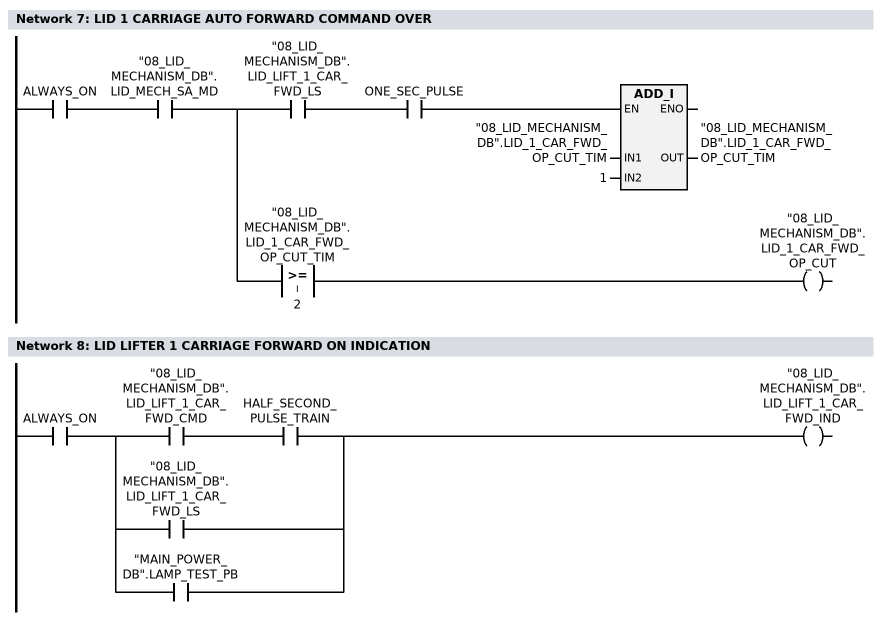
[picture p120: LID_1_MECHANISM networks 7-8]
NETWORK
TITLE = LID 1 CARRIAGE AUTO FORWARD COMMAND OVER
      A     "ALWAYS_ON";
      A     "08_LID_MECHANISM_DB".LID_MECH_SA_MD;
      =     L 0.0;
      A     L 0.0;
      A     "08_LID_MECHANISM_DB".LID_LIFT_1_CAR_FWD_LS;
      A     "ONE_SEC_PULSE";
      JNB   _002;
      L     "08_LID_MECHANISM_DB".LID_1_CAR_FWD_OP_CUT_TIM;
      L     1;
      +I;
      T     "08_LID_MECHANISM_DB".LID_1_CAR_FWD_OP_CUT_TIM;
_002: NOP   0;
      A     L 0.0;
      A(;
      L     "08_LID_MECHANISM_DB".LID_1_CAR_FWD_OP_CUT_TIM;
      L     2;
      >=I;
      );
      =     "08_LID_MECHANISM_DB".LID_1_CAR_FWD_OP_CUT;
NETWORK
TITLE = LID LIFTER 1 CARRIAGE FORWARD ON INDICATION
      A     "ALWAYS_ON";
      A(;
      A     "08_LID_MECHANISM_DB".LID_LIFT_1_CAR_FWD_CMD;
      A     "HALF_SECOND_PULSE_TRAIN";
      O     "08_LID_MECHANISM_DB".LID_LIFT_1_CAR_FWD_LS;
      O     "MAIN_POWER_DB".LAMP_TEST_PB;
      );
      =     "08_LID_MECHANISM_DB".LID_LIFT_1_CAR_FWD_IND;
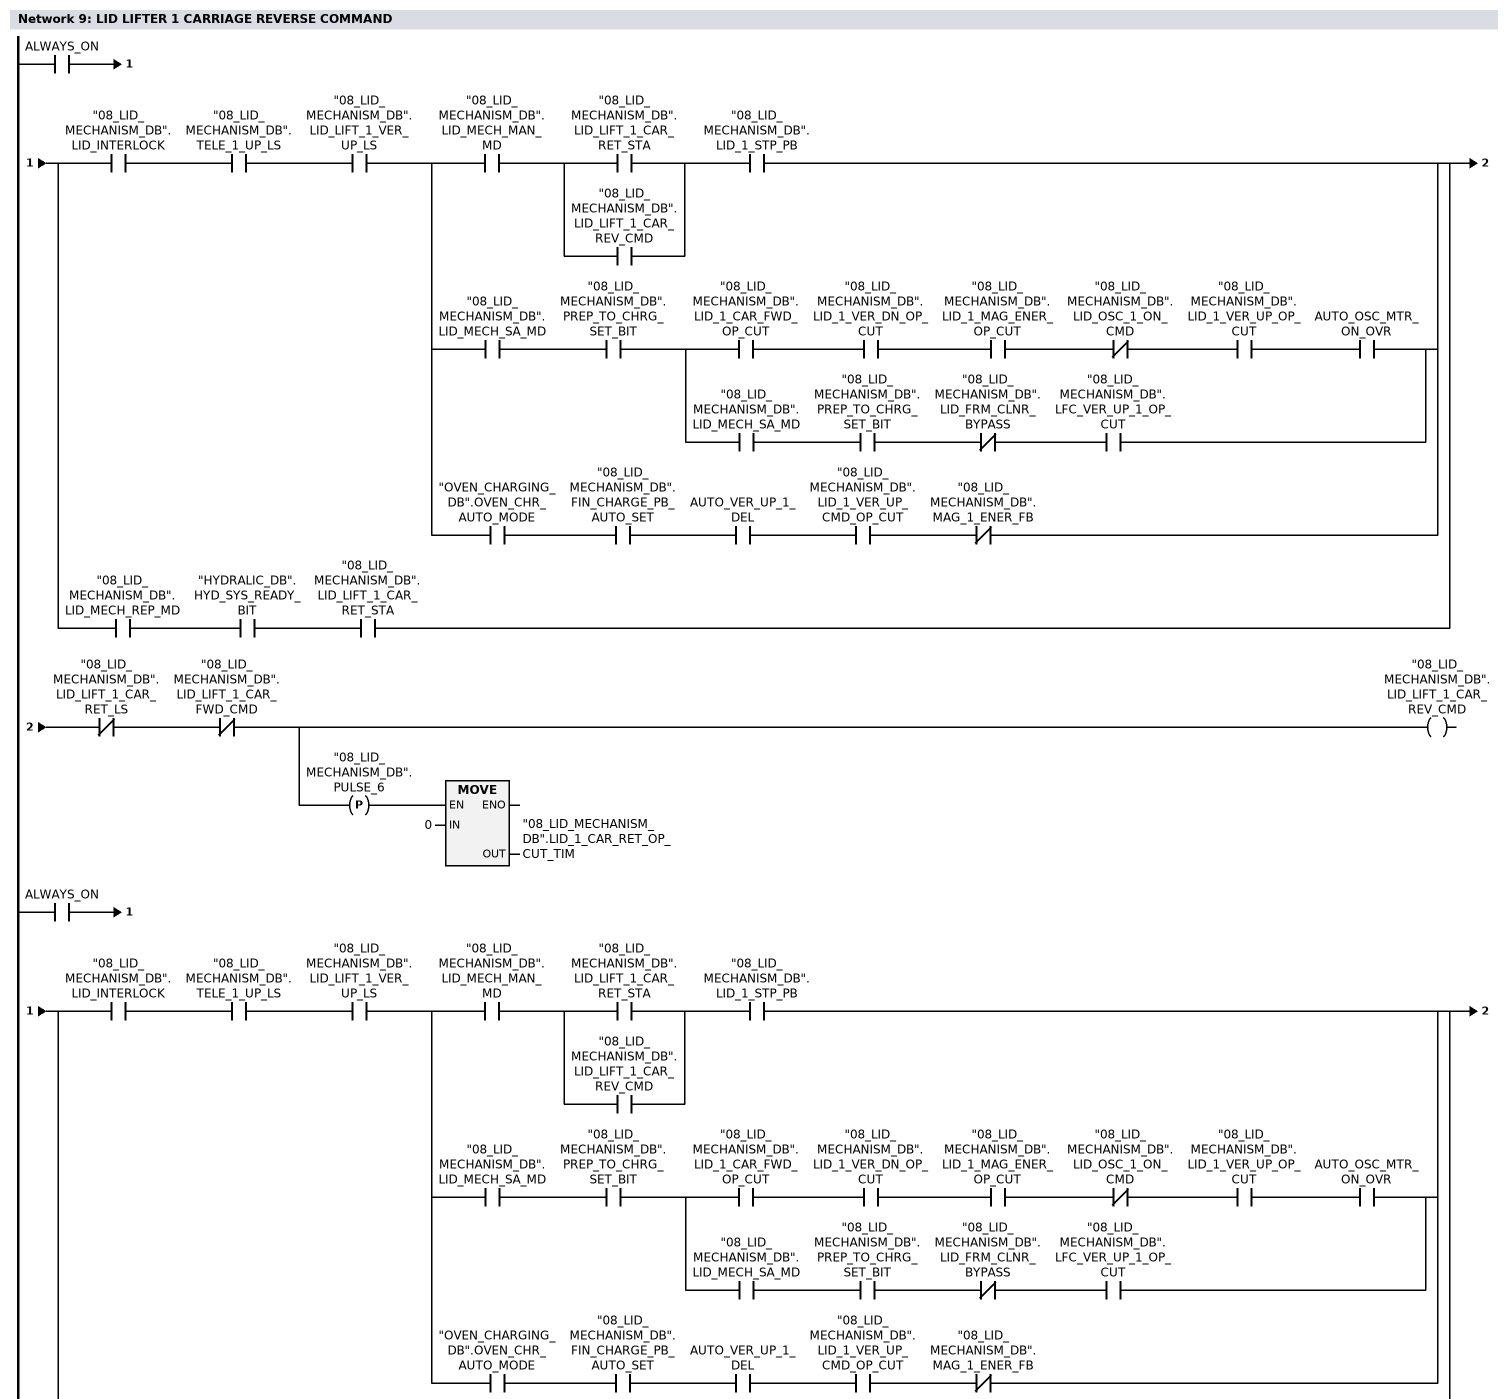
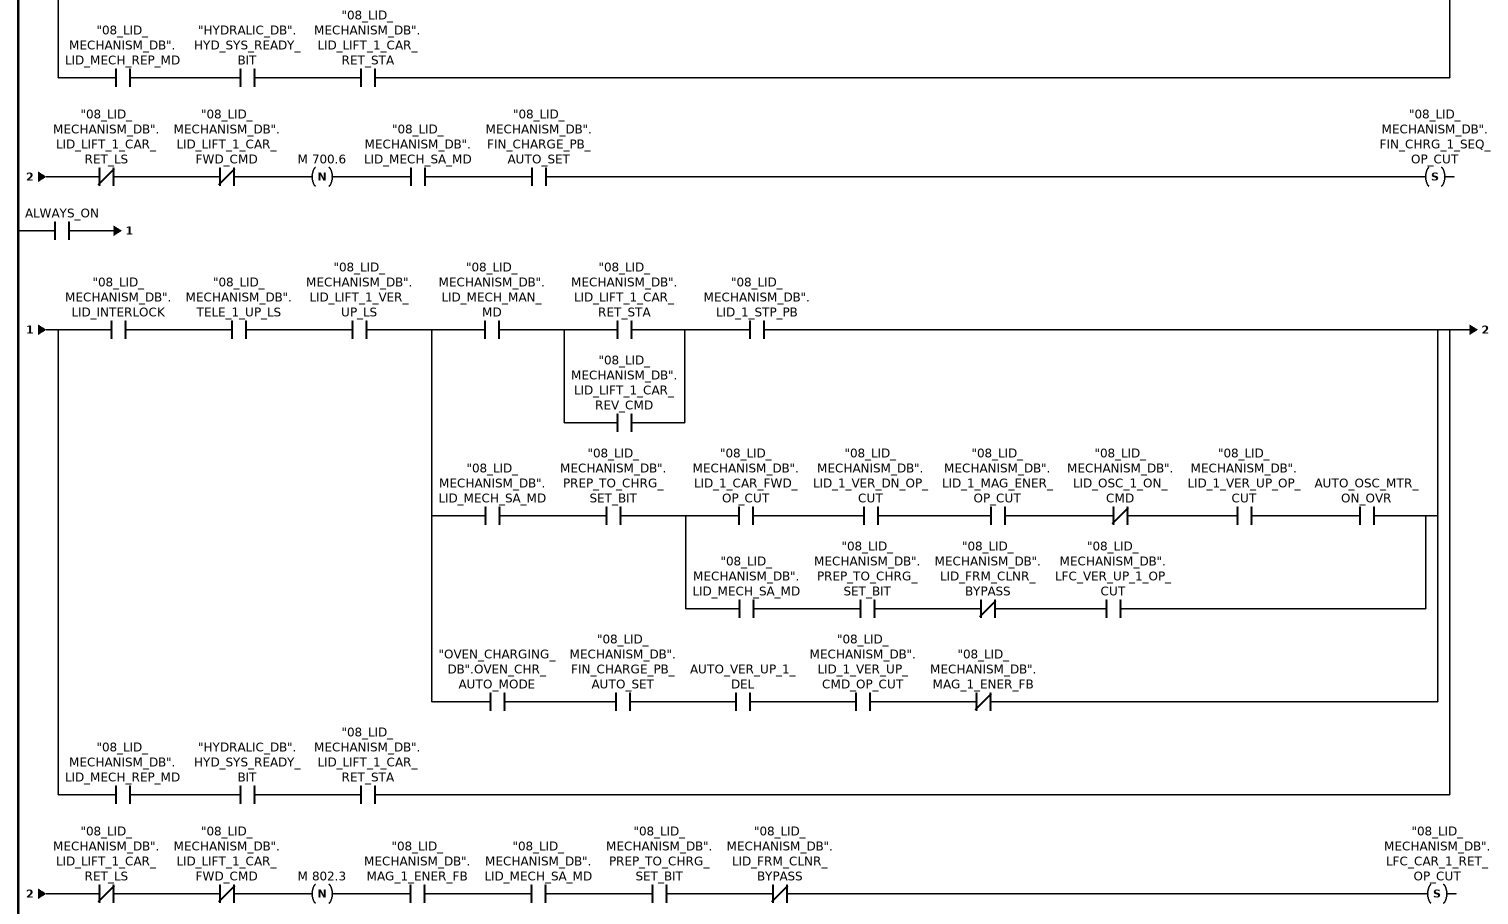
NETWORK
TITLE = LID LIFTER 1 CARRIAGE REVERSE COMMAND
      A     "ALWAYS_ON";
      A(;
      A     "08_LID_MECHANISM_DB".LID_INTERLOCK;
      A     "08_LID_MECHANISM_DB".TELE_1_UP_LS;
      A     "08_LID_MECHANISM_DB".LID_LIFT_1_VER_UP_LS;
      A(;
      A     "08_LID_MECHANISM_DB".LID_MECH_MAN_MD;
      A(;
      O     "08_LID_MECHANISM_DB".LID_LIFT_1_CAR_RET_STA;
      O     "08_LID_MECHANISM_DB".LID_LIFT_1_CAR_REV_CMD;
      );
      A     "08_LID_MECHANISM_DB".LID_1_STP_PB;
      O;
      A     "08_LID_MECHANISM_DB".LID_MECH_SA_MD;
      A     "08_LID_MECHANISM_DB".PREP_TO_CHRG_SET_BIT;
      A(;
      A     "08_LID_MECHANISM_DB".LID_1_CAR_FWD_OP_CUT;
      A     "08_LID_MECHANISM_DB".LID_1_VER_DN_OP_CUT;
      A     "08_LID_MECHANISM_DB".LID_1_MAG_ENER_OP_CUT;
      AN    "08_LID_MECHANISM_DB".LID_OSC_1_ON_CMD;
      A     "08_LID_MECHANISM_DB".LID_1_VER_UP_OP_CUT;
      A     "AUTO_OSC_MTR_ON_OVR";
      O;
      A     "08_LID_MECHANISM_DB".LID_MECH_SA_MD;
      A     "08_LID_MECHANISM_DB".PREP_TO_CHRG_SET_BIT;
      AN    "08_LID_MECHANISM_DB".LID_FRM_CLNR_BYPASS;
      A     "08_LID_MECHANISM_DB".LFC_VER_UP_1_OP_CUT;
      );
      O;
      A     "OVEN_CHARGING_DB".OVEN_CHR_AUTO_MODE;
      A     "08_LID_MECHANISM_DB".FIN_CHARGE_PB_AUTO_SET;
      A     "AUTO_VER_UP_1_DEL";
      A     "08_LID_MECHANISM_DB".LID_1_VER_UP_CMD_OP_CUT;
      AN    "08_LID_MECHANISM_DB".MAG_1_ENER_FB;
      );
      O;
      A     "08_LID_MECHANISM_DB".LID_MECH_REP_MD;
      A     "HYDRALIC_DB".HYD_SYS_READY_BIT;
      A     "08_LID_MECHANISM_DB".LID_LIFT_1_CAR_RET_STA;
      );
      AN    "08_LID_MECHANISM_DB".LID_LIFT_1_CAR_RET_LS;
      AN    "08_LID_MECHANISM_DB".LID_LIFT_1_CAR_FWD_CMD;
      =     L 0.0;
      A     L 0.0;
      BLD   102;
      =     "08_LID_MECHANISM_DB".LID_LIFT_1_CAR_REV_CMD;
      A     L 0.0;
      FP    "08_LID_MECHANISM_DB".PULSE_6;
      JNB   _003;
      L     0;
      T     "08_LID_MECHANISM_DB".LID_1_CAR_RET_OP_CUT_TIM;
_003: NOP   0;
      A(;
      A     L 0.0;
      FN    M 700.6;
      );
      A     "08_LID_MECHANISM_DB".LID_MECH_SA_MD;
      A     "08_LID_MECHANISM_DB".FIN_CHARGE_PB_AUTO_SET;
      S     "08_LID_MECHANISM_DB".FIN_CHRG_1_SEQ_OP_CUT;
      A(;
      A     L 0.0;
      FN    M 802.3;
      );
      A     "08_LID_MECHANISM_DB".MAG_1_ENER_FB;
      A     "08_LID_MECHANISM_DB".LID_MECH_SA_MD;
      A     "08_LID_MECHANISM_DB".PREP_TO_CHRG_SET_BIT;
      AN    "08_LID_MECHANISM_DB".LID_FRM_CLNR_BYPASS;
      S     "08_LID_MECHANISM_DB".LFC_CAR_1_RET_OP_CUT;
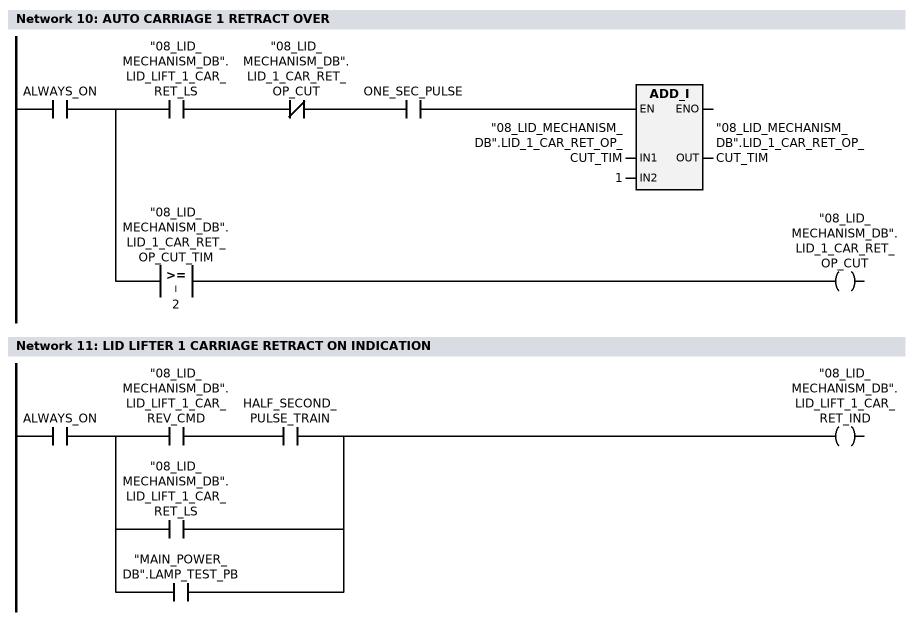
NETWORK
TITLE = AUTO CARRIAGE 1 RETRACT OVER
      A     "ALWAYS_ON";
      =     L 0.0;
      A     L 0.0;
      A     "08_LID_MECHANISM_DB".LID_LIFT_1_CAR_RET_LS;
      AN    "08_LID_MECHANISM_DB".LID_1_CAR_RET_OP_CUT;
      A     "ONE_SEC_PULSE";
      JNB   _004;
      L     "08_LID_MECHANISM_DB".LID_1_CAR_RET_OP_CUT_TIM;
      L     1;
      +I;
      T     "08_LID_MECHANISM_DB".LID_1_CAR_RET_OP_CUT_TIM;
_004: NOP   0;
      A     L 0.0;
      A(;
      L     "08_LID_MECHANISM_DB".LID_1_CAR_RET_OP_CUT_TIM;
      L     2;
      >=I;
      );
      =     "08_LID_MECHANISM_DB".LID_1_CAR_RET_OP_CUT;
NETWORK
TITLE = LID LIFTER 1 CARRIAGE RETRACT ON INDICATION
      A     "ALWAYS_ON";
      A(;
      A     "08_LID_MECHANISM_DB".LID_LIFT_1_CAR_REV_CMD;
      A     "HALF_SECOND_PULSE_TRAIN";
      O     "08_LID_MECHANISM_DB".LID_LIFT_1_CAR_RET_LS;
      O     "MAIN_POWER_DB".LAMP_TEST_PB;
      );
      =     "08_LID_MECHANISM_DB".LID_LIFT_1_CAR_RET_IND;
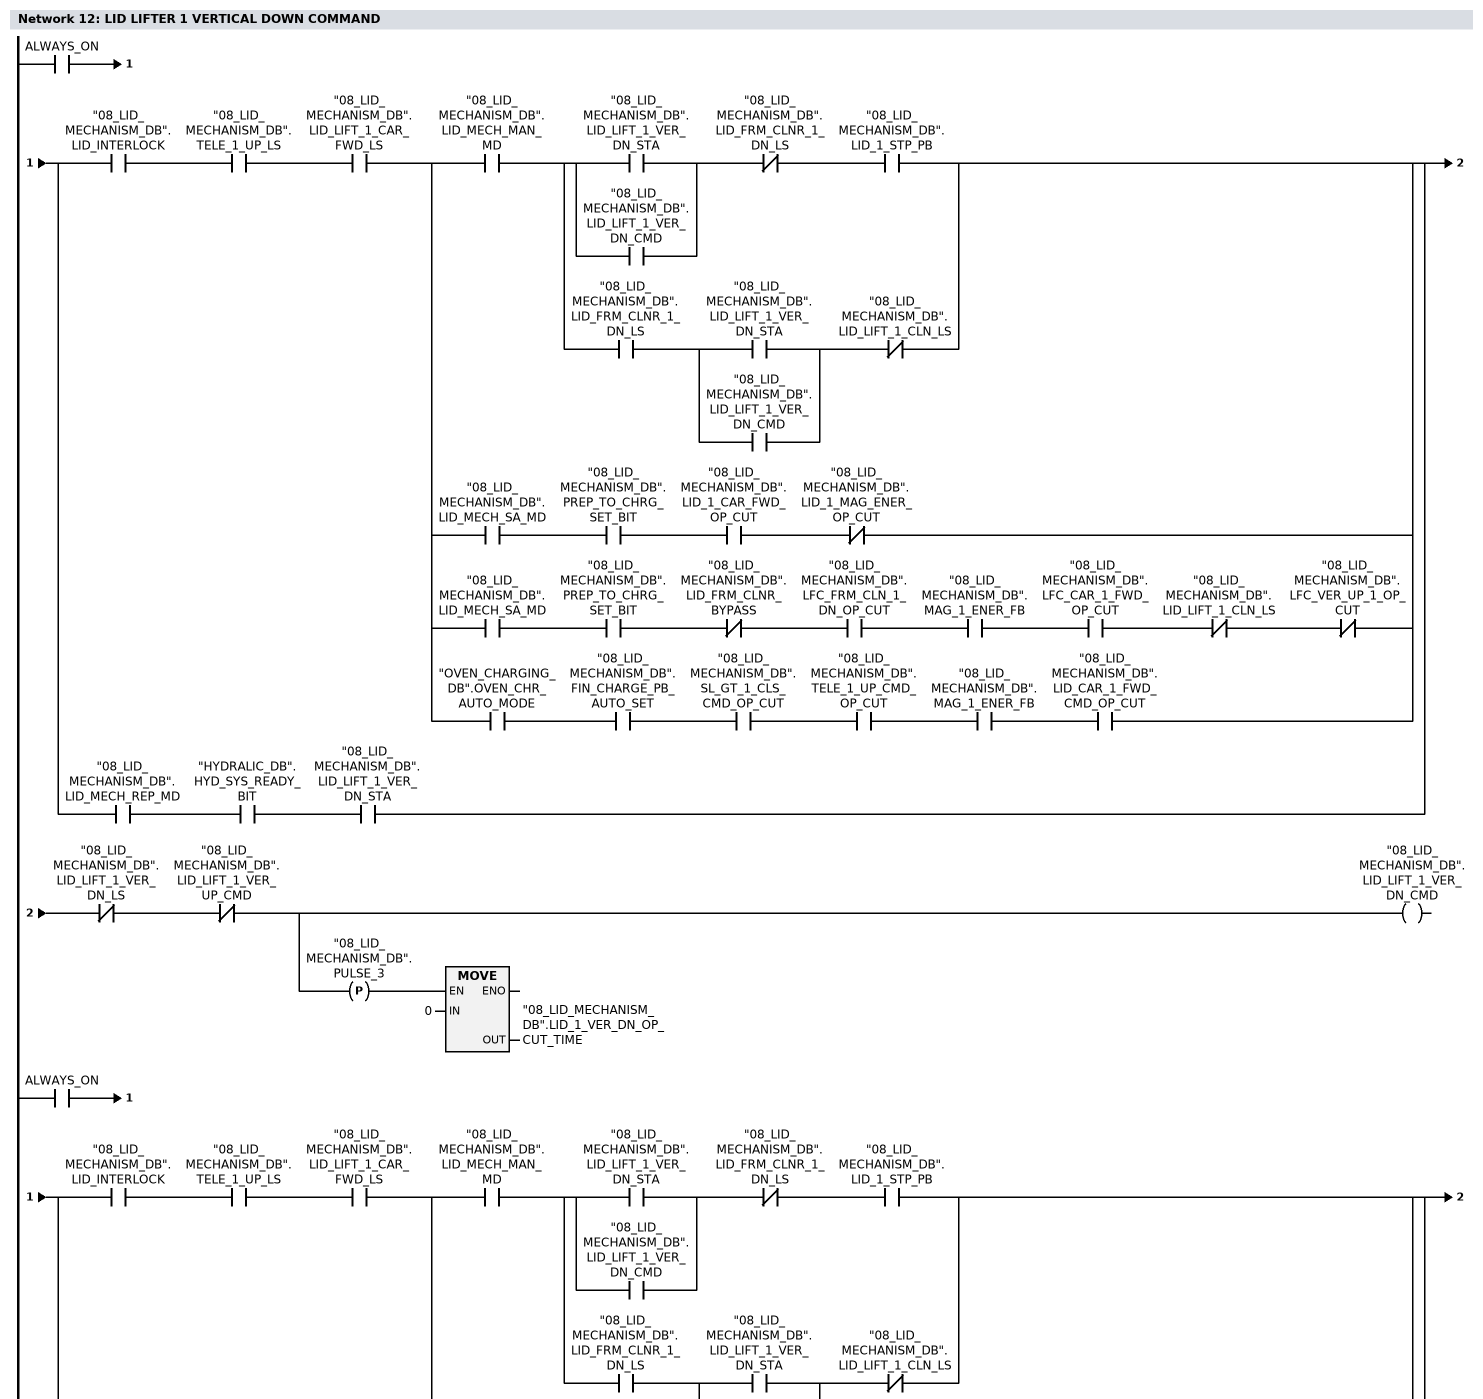
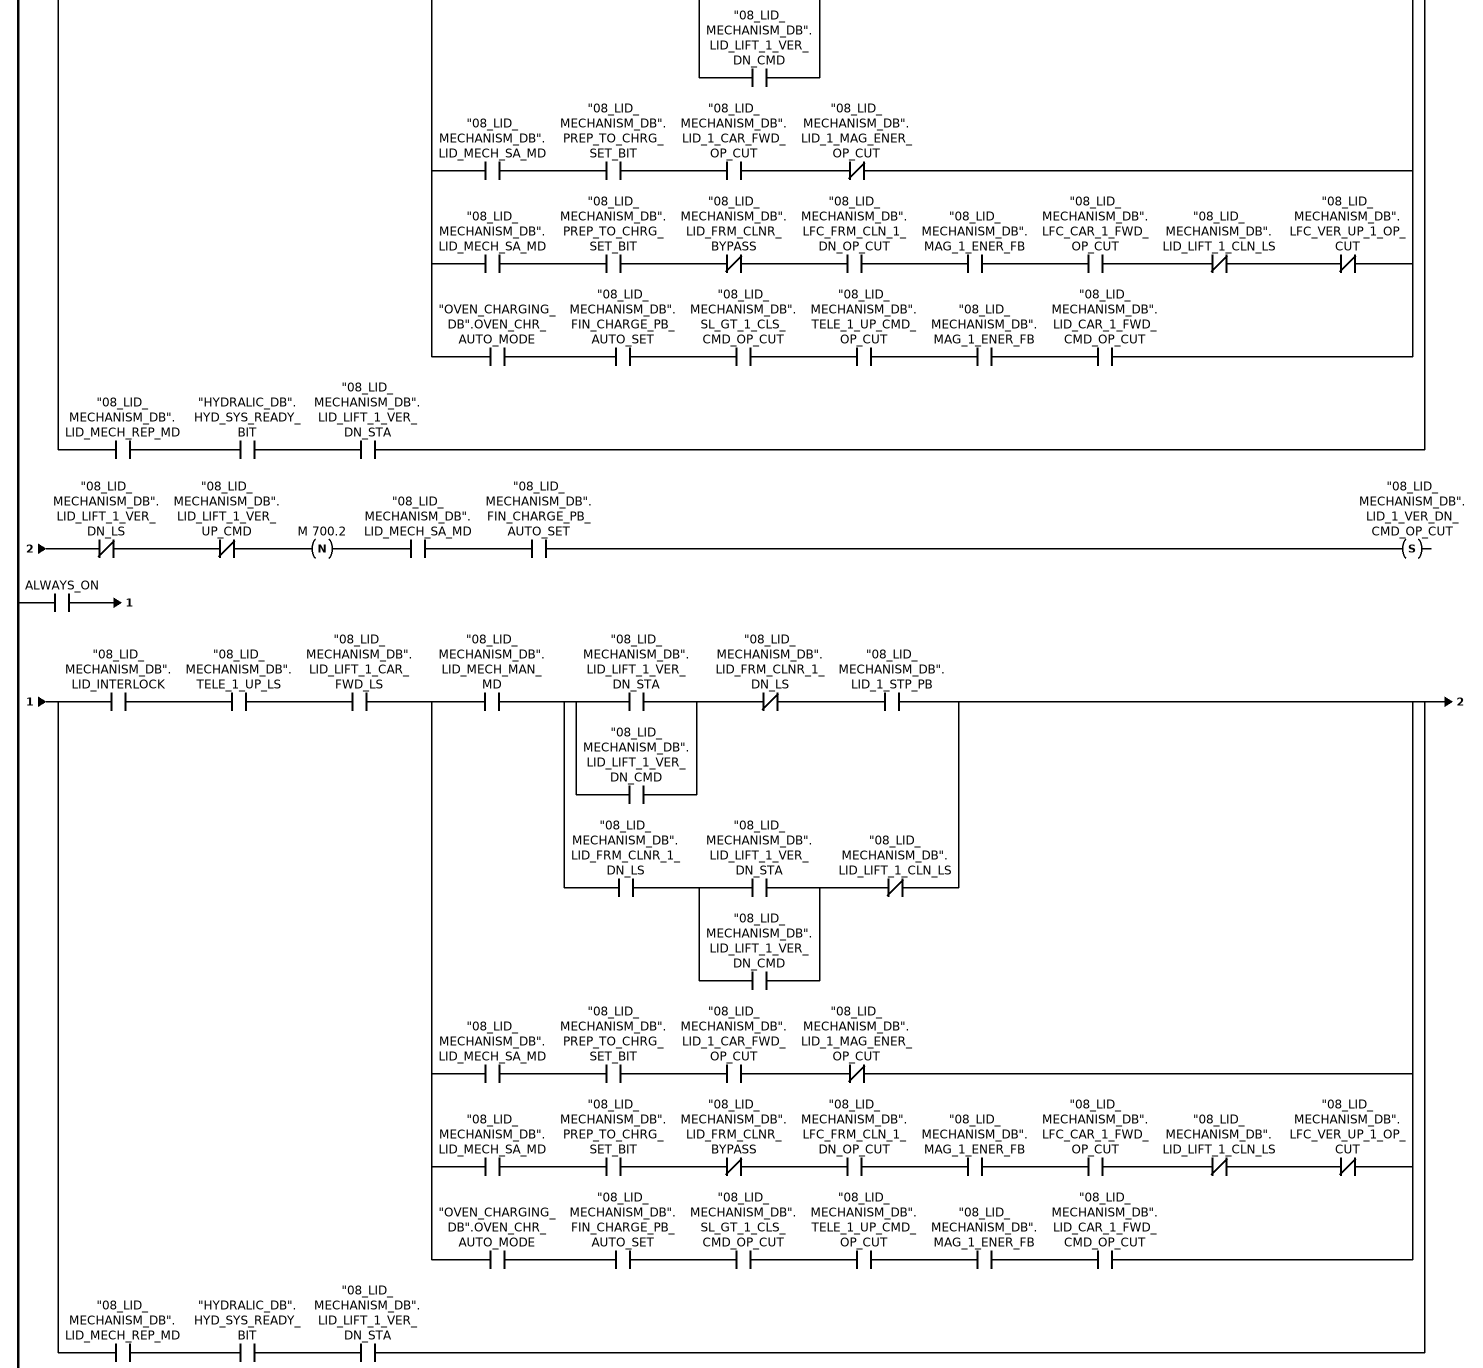
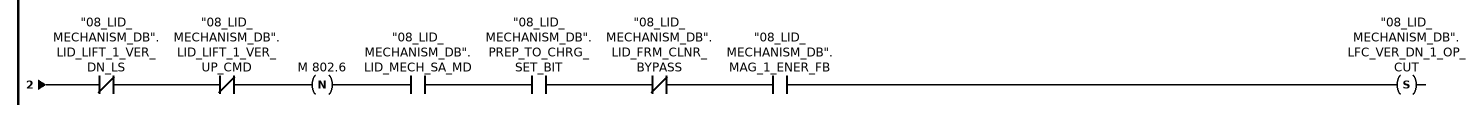
NETWORK
TITLE = LID LIFTER 1 VERTICAL DOWN COMMAND
      A     "ALWAYS_ON";
      A(;
      A     "08_LID_MECHANISM_DB".LID_INTERLOCK;
      A     "08_LID_MECHANISM_DB".TELE_1_UP_LS;
      A     "08_LID_MECHANISM_DB".LID_LIFT_1_CAR_FWD_LS;
      A(;
      A     "08_LID_MECHANISM_DB".LID_MECH_MAN_MD;
      A(;
      A(;
      O     "08_LID_MECHANISM_DB".LID_LIFT_1_VER_DN_STA;
      O     "08_LID_MECHANISM_DB".LID_LIFT_1_VER_DN_CMD;
      );
      AN    "08_LID_MECHANISM_DB".LID_FRM_CLNR_1_DN_LS;
      A     "08_LID_MECHANISM_DB".LID_1_STP_PB;
      O;
      A     "08_LID_MECHANISM_DB".LID_FRM_CLNR_1_DN_LS;
      A(;
      O     "08_LID_MECHANISM_DB".LID_LIFT_1_VER_DN_STA;
      O     "08_LID_MECHANISM_DB".LID_LIFT_1_VER_DN_CMD;
      );
      AN    "08_LID_MECHANISM_DB".LID_LIFT_1_CLN_LS;
      );
      O;
      A     "08_LID_MECHANISM_DB".LID_MECH_SA_MD;
      A     "08_LID_MECHANISM_DB".PREP_TO_CHRG_SET_BIT;
      A     "08_LID_MECHANISM_DB".LID_1_CAR_FWD_OP_CUT;
      AN    "08_LID_MECHANISM_DB".LID_1_MAG_ENER_OP_CUT;
      O;
      A     "08_LID_MECHANISM_DB".LID_MECH_SA_MD;
      A     "08_LID_MECHANISM_DB".PREP_TO_CHRG_SET_BIT;
      AN    "08_LID_MECHANISM_DB".LID_FRM_CLNR_BYPASS;
      A     "08_LID_MECHANISM_DB".LFC_FRM_CLN_1_DN_OP_CUT;
      A     "08_LID_MECHANISM_DB".MAG_1_ENER_FB;
      A     "08_LID_MECHANISM_DB".LFC_CAR_1_FWD_OP_CUT;
      AN    "08_LID_MECHANISM_DB".LID_LIFT_1_CLN_LS;
      AN    "08_LID_MECHANISM_DB".LFC_VER_UP_1_OP_CUT;
      O;
      A     "OVEN_CHARGING_DB".OVEN_CHR_AUTO_MODE;
      A     "08_LID_MECHANISM_DB".FIN_CHARGE_PB_AUTO_SET;
      A     "08_LID_MECHANISM_DB".SL_GT_1_CLS_CMD_OP_CUT;
      A     "08_LID_MECHANISM_DB".TELE_1_UP_CMD_OP_CUT;
      A     "08_LID_MECHANISM_DB".MAG_1_ENER_FB;
      A     "08_LID_MECHANISM_DB".LID_CAR_1_FWD_CMD_OP_CUT;
      );
      O;
      A     "08_LID_MECHANISM_DB".LID_MECH_REP_MD;
      A     "HYDRALIC_DB".HYD_SYS_READY_BIT;
      A     "08_LID_MECHANISM_DB".LID_LIFT_1_VER_DN_STA;
      );
      AN    "08_LID_MECHANISM_DB".LID_LIFT_1_VER_DN_LS;
      AN    "08_LID_MECHANISM_DB".LID_LIFT_1_VER_UP_CMD;
      =     L 0.0;
      A     L 0.0;
      BLD   102;
      =     "08_LID_MECHANISM_DB".LID_LIFT_1_VER_DN_CMD;
      A     L 0.0;
      FP    "08_LID_MECHANISM_DB".PULSE_3;
      JNB   _005;
      L     0;
      T     "08_LID_MECHANISM_DB".LID_1_VER_DN_OP_CUT_TIME;
_005: NOP   0;
      A(;
      A     L 0.0;
      FN    M 700.2;
      );
      A     "08_LID_MECHANISM_DB".LID_MECH_SA_MD;
      A     "08_LID_MECHANISM_DB".FIN_CHARGE_PB_AUTO_SET;
      S     "08_LID_MECHANISM_DB".LID_1_VER_DN_CMD_OP_CUT;
      A(;
      A     L 0.0;
      FN    M 802.6;
      );
      A     "08_LID_MECHANISM_DB".LID_MECH_SA_MD;
      A     "08_LID_MECHANISM_DB".PREP_TO_CHRG_SET_BIT;
      AN    "08_LID_MECHANISM_DB".LID_FRM_CLNR_BYPASS;
      A     "08_LID_MECHANISM_DB".MAG_1_ENER_FB;
      S     "08_LID_MECHANISM_DB".LFC_VER_DN_1_OP_CUT;
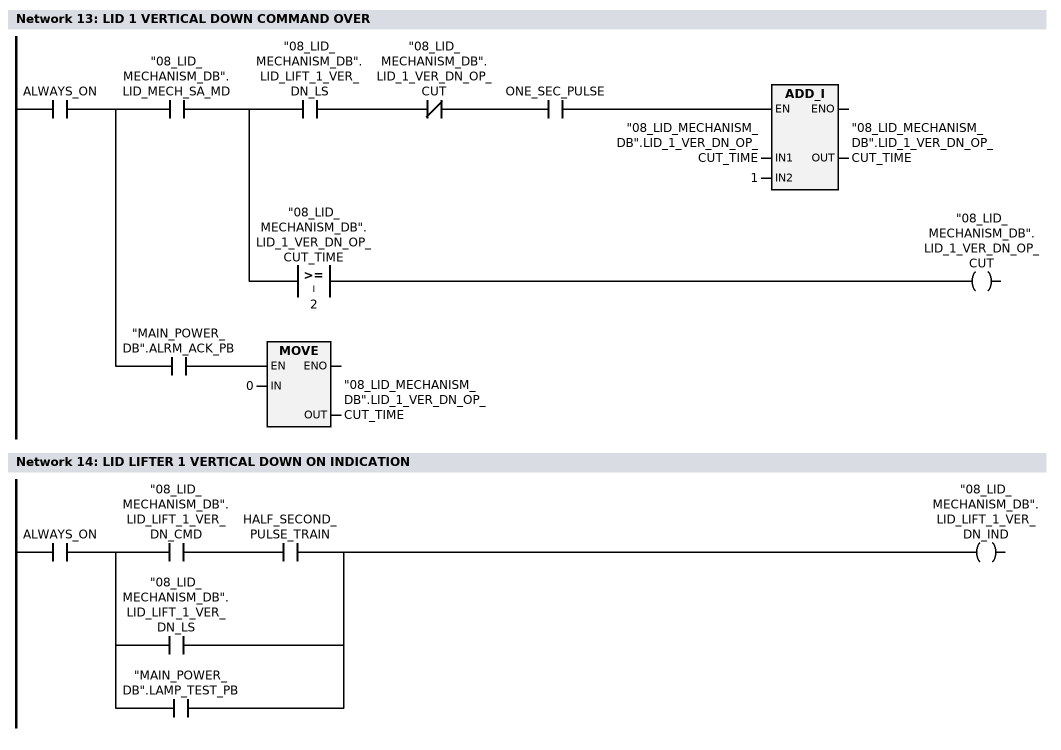
NETWORK
TITLE = LID 1 VERTICAL DOWN COMMAND OVER
      A     "ALWAYS_ON";
      =     L 0.0;
      A     L 0.0;
      A     "08_LID_MECHANISM_DB".LID_MECH_SA_MD;
      =     L 0.1;
      A     L 0.1;
      A     "08_LID_MECHANISM_DB".LID_LIFT_1_VER_DN_LS;
      AN    "08_LID_MECHANISM_DB".LID_1_VER_DN_OP_CUT;
      A     "ONE_SEC_PULSE";
      JNB   _006;
      L     "08_LID_MECHANISM_DB".LID_1_VER_DN_OP_CUT_TIME;
      L     1;
      +I;
      T     "08_LID_MECHANISM_DB".LID_1_VER_DN_OP_CUT_TIME;
_006: NOP   0;
      A     L 0.1;
      A(;
      L     "08_LID_MECHANISM_DB".LID_1_VER_DN_OP_CUT_TIME;
      L     2;
      >=I;
      );
      =     "08_LID_MECHANISM_DB".LID_1_VER_DN_OP_CUT;
      A     L 0.0;
      A     "MAIN_POWER_DB".ALRM_ACK_PB;
      JNB   _007;
      L     0;
      T     "08_LID_MECHANISM_DB".LID_1_VER_DN_OP_CUT_TIME;
_007: NOP   0;
NETWORK
TITLE = LID LIFTER 1 VERTICAL DOWN ON INDICATION
      A     "ALWAYS_ON";
      A(;
      A     "08_LID_MECHANISM_DB".LID_LIFT_1_VER_DN_CMD;
      A     "HALF_SECOND_PULSE_TRAIN";
      O     "08_LID_MECHANISM_DB".LID_LIFT_1_VER_DN_LS;
      O     "MAIN_POWER_DB".LAMP_TEST_PB;
      );
      =     "08_LID_MECHANISM_DB".LID_LIFT_1_VER_DN_IND;
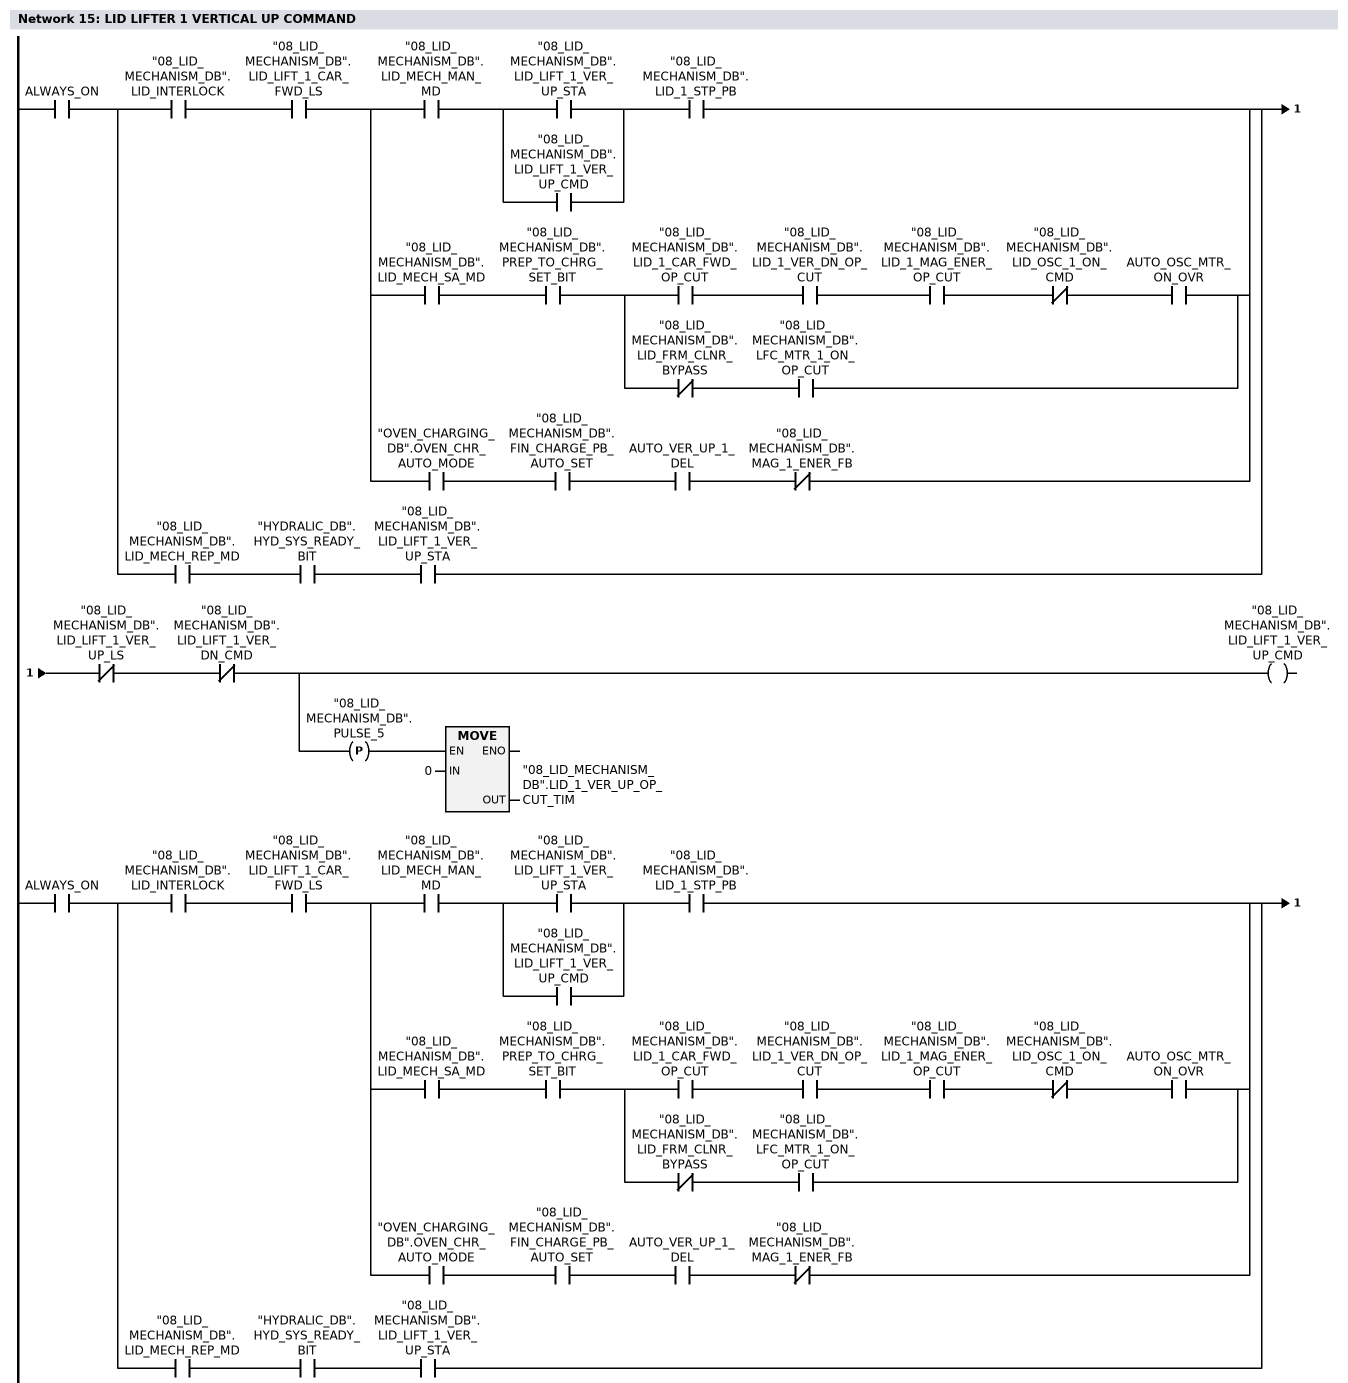
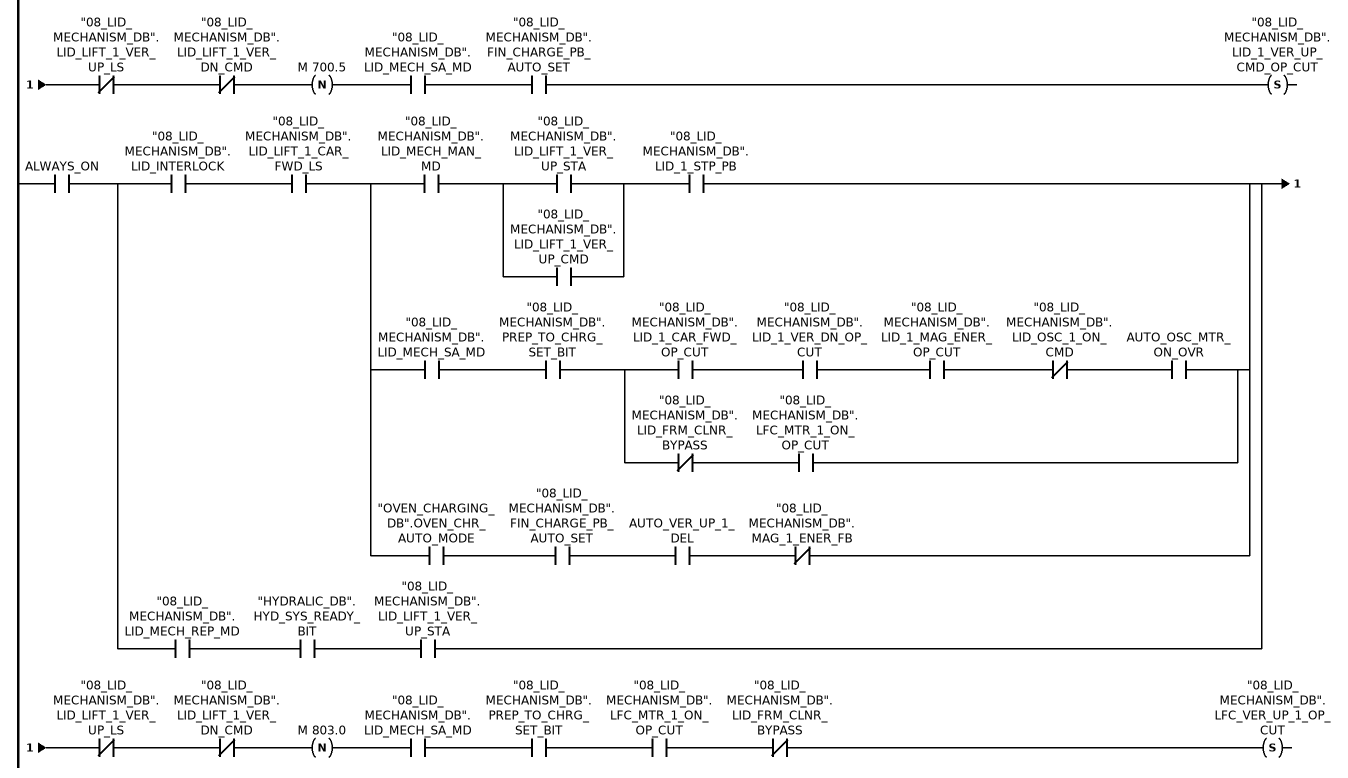
NETWORK
TITLE = LID LIFTER 1 VERTICAL UP COMMAND
      A     "ALWAYS_ON";
      A(;
      A     "08_LID_MECHANISM_DB".LID_INTERLOCK;
      A     "08_LID_MECHANISM_DB".LID_LIFT_1_CAR_FWD_LS;
      A(;
      A     "08_LID_MECHANISM_DB".LID_MECH_MAN_MD;
      A(;
      O     "08_LID_MECHANISM_DB".LID_LIFT_1_VER_UP_STA;
      O     "08_LID_MECHANISM_DB".LID_LIFT_1_VER_UP_CMD;
      );
      A     "08_LID_MECHANISM_DB".LID_1_STP_PB;
      O;
      A     "08_LID_MECHANISM_DB".LID_MECH_SA_MD;
      A     "08_LID_MECHANISM_DB".PREP_TO_CHRG_SET_BIT;
      A(;
      A     "08_LID_MECHANISM_DB".LID_1_CAR_FWD_OP_CUT;
      A     "08_LID_MECHANISM_DB".LID_1_VER_DN_OP_CUT;
      A     "08_LID_MECHANISM_DB".LID_1_MAG_ENER_OP_CUT;
      AN    "08_LID_MECHANISM_DB".LID_OSC_1_ON_CMD;
      A     "AUTO_OSC_MTR_ON_OVR";
      O;
      AN    "08_LID_MECHANISM_DB".LID_FRM_CLNR_BYPASS;
      A     "08_LID_MECHANISM_DB".LFC_MTR_1_ON_OP_CUT;
      );
      O;
      A     "OVEN_CHARGING_DB".OVEN_CHR_AUTO_MODE;
      A     "08_LID_MECHANISM_DB".FIN_CHARGE_PB_AUTO_SET;
      A     "AUTO_VER_UP_1_DEL";
      AN    "08_LID_MECHANISM_DB".MAG_1_ENER_FB;
      );
      O;
      A     "08_LID_MECHANISM_DB".LID_MECH_REP_MD;
      A     "HYDRALIC_DB".HYD_SYS_READY_BIT;
      A     "08_LID_MECHANISM_DB".LID_LIFT_1_VER_UP_STA;
      );
      AN    "08_LID_MECHANISM_DB".LID_LIFT_1_VER_UP_LS;
      AN    "08_LID_MECHANISM_DB".LID_LIFT_1_VER_DN_CMD;
      =     L 0.0;
      A     L 0.0;
      BLD   102;
      =     "08_LID_MECHANISM_DB".LID_LIFT_1_VER_UP_CMD;
      A     L 0.0;
      FP    "08_LID_MECHANISM_DB".PULSE_5;
      JNB   _008;
      L     0;
      T     "08_LID_MECHANISM_DB".LID_1_VER_UP_OP_CUT_TIM;
_008: NOP   0;
      A(;
      A     L 0.0;
      FN    M 700.5;
      );
      A     "08_LID_MECHANISM_DB".LID_MECH_SA_MD;
      A     "08_LID_MECHANISM_DB".FIN_CHARGE_PB_AUTO_SET;
      S     "08_LID_MECHANISM_DB".LID_1_VER_UP_CMD_OP_CUT;
      A(;
      A     L 0.0;
      FN    M 803.0;
      );
      A     "08_LID_MECHANISM_DB".LID_MECH_SA_MD;
      A     "08_LID_MECHANISM_DB".PREP_TO_CHRG_SET_BIT;
      A     "08_LID_MECHANISM_DB".LFC_MTR_1_ON_OP_CUT;
      AN    "08_LID_MECHANISM_DB".LID_FRM_CLNR_BYPASS;
      S     "08_LID_MECHANISM_DB".LFC_VER_UP_1_OP_CUT;
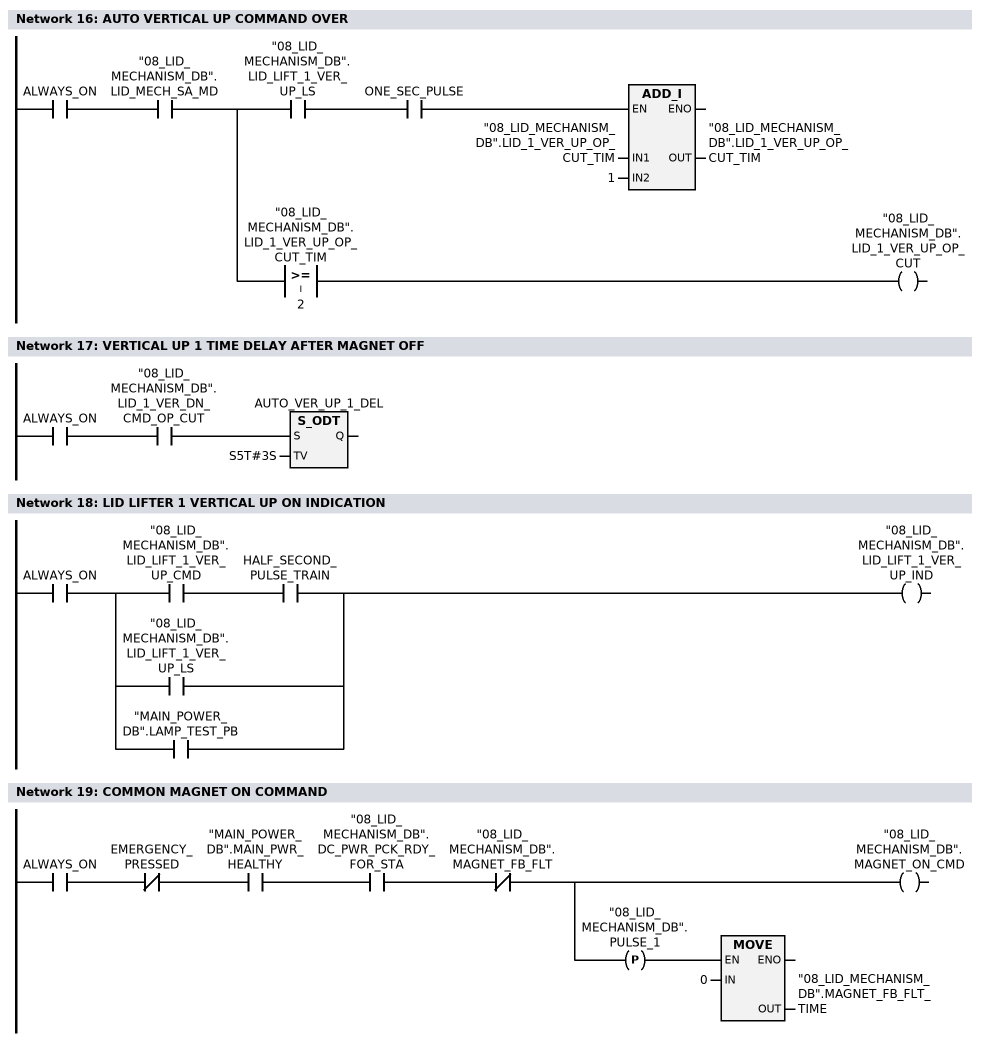
NETWORK
TITLE = AUTO VERTICAL UP COMMAND OVER
      A     "ALWAYS_ON";
      A     "08_LID_MECHANISM_DB".LID_MECH_SA_MD;
      =     L 0.0;
      A     L 0.0;
      A     "08_LID_MECHANISM_DB".LID_LIFT_1_VER_UP_LS;
      A     "ONE_SEC_PULSE";
      JNB   _009;
      L     "08_LID_MECHANISM_DB".LID_1_VER_UP_OP_CUT_TIM;
      L     1;
      +I;
      T     "08_LID_MECHANISM_DB".LID_1_VER_UP_OP_CUT_TIM;
_009: NOP   0;
      A     L 0.0;
      A(;
      L     "08_LID_MECHANISM_DB".LID_1_VER_UP_OP_CUT_TIM;
      L     2;
      >=I;
      );
      =     "08_LID_MECHANISM_DB".LID_1_VER_UP_OP_CUT;
NETWORK
TITLE = VERTICAL UP 1 TIME DELAY AFTER MAGNET OFF
      A     "ALWAYS_ON";
      A     "08_LID_MECHANISM_DB".LID_1_VER_DN_CMD_OP_CUT;
      L     S5T#3S;
      SD    "AUTO_VER_UP_1_DEL";
      NOP   0;
      NOP   0;
      NOP   0;
      NOP   0;
NETWORK
TITLE = LID LIFTER 1 VERTICAL UP ON INDICATION
      A     "ALWAYS_ON";
      A(;
      A     "08_LID_MECHANISM_DB".LID_LIFT_1_VER_UP_CMD;
      A     "HALF_SECOND_PULSE_TRAIN";
      O     "08_LID_MECHANISM_DB".LID_LIFT_1_VER_UP_LS;
      O     "MAIN_POWER_DB".LAMP_TEST_PB;
      );
      =     "08_LID_MECHANISM_DB".LID_LIFT_1_VER_UP_IND;
NETWORK
TITLE = COMMON MAGNET ON COMMAND
      A     "ALWAYS_ON";
      AN    "EMERGENCY_PRESSED";
      A     "MAIN_POWER_DB".MAIN_PWR_HEALTHY;
      A     "08_LID_MECHANISM_DB".DC_PWR_PCK_RDY_FOR_STA;
      AN    "08_LID_MECHANISM_DB".MAGNET_FB_FLT;
      =     L 0.0;
      A     L 0.0;
      BLD   102;
      =     "08_LID_MECHANISM_DB".MAGNET_ON_CMD;
      A     L 0.0;
      FP    "08_LID_MECHANISM_DB".PULSE_1;
      JNB   _00a;
      L     0;
      T     "08_LID_MECHANISM_DB".MAGNET_FB_FLT_TIME;
_00a: NOP   0;
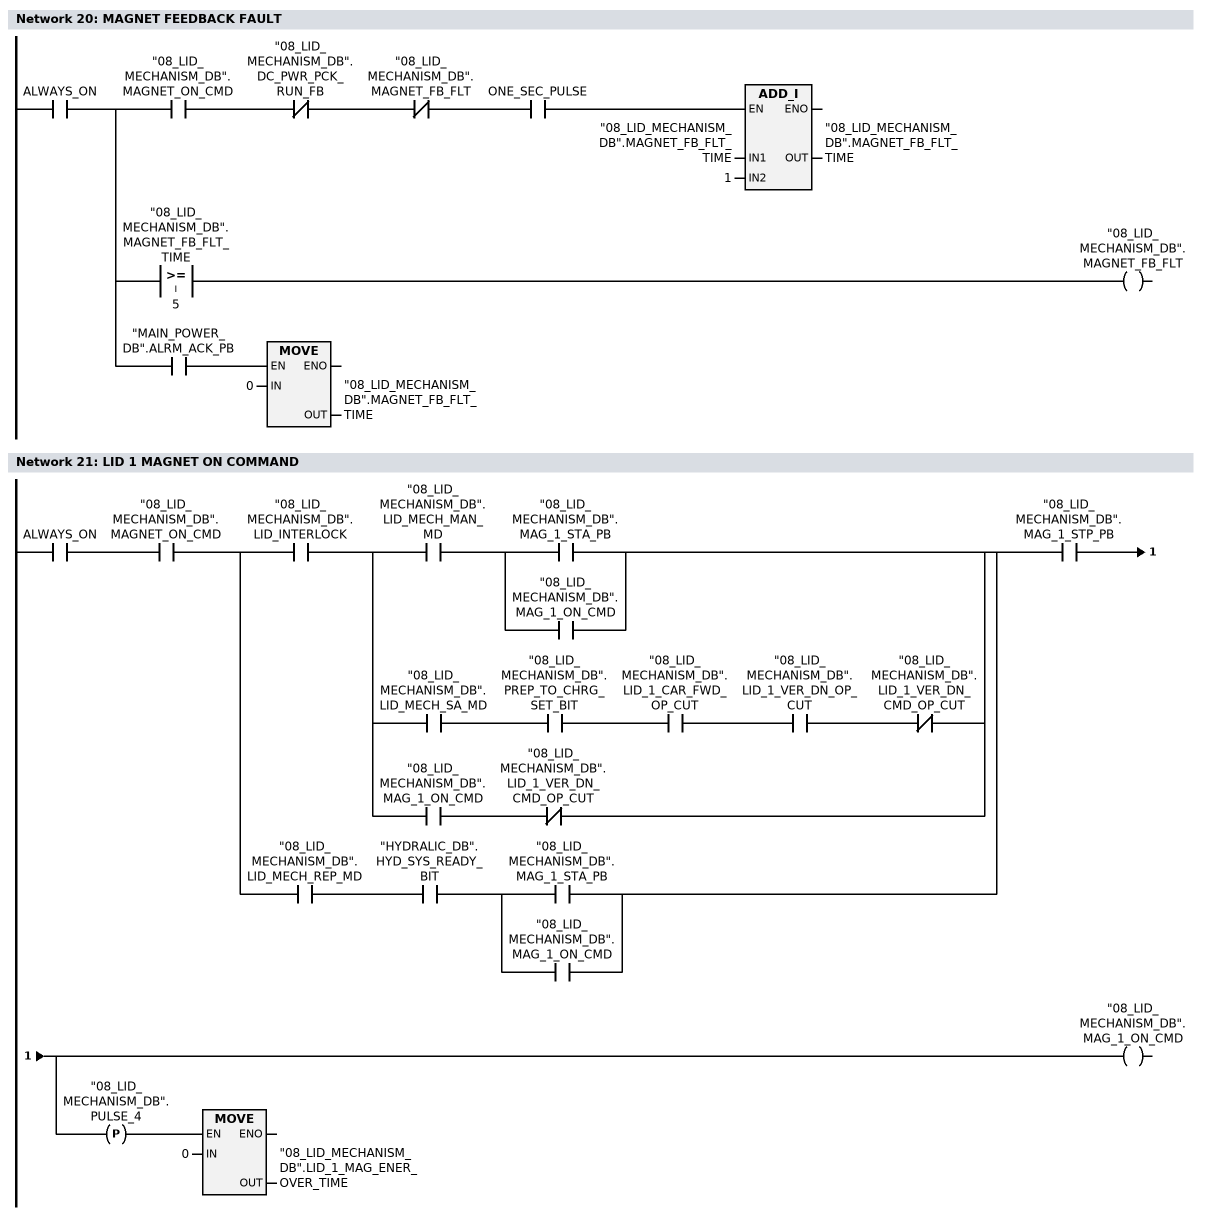
NETWORK
TITLE = MAGNET FEEDBACK FAULT
      A     "ALWAYS_ON";
      =     L 0.0;
      A     L 0.0;
      A     "08_LID_MECHANISM_DB".MAGNET_ON_CMD;
      AN    "08_LID_MECHANISM_DB".DC_PWR_PCK_RUN_FB;
      AN    "08_LID_MECHANISM_DB".MAGNET_FB_FLT;
      A     "ONE_SEC_PULSE";
      JNB   _00b;
      L     "08_LID_MECHANISM_DB".MAGNET_FB_FLT_TIME;
      L     1;
      +I;
      T     "08_LID_MECHANISM_DB".MAGNET_FB_FLT_TIME;
_00b: NOP   0;
      A     L 0.0;
      A(;
      L     "08_LID_MECHANISM_DB".MAGNET_FB_FLT_TIME;
      L     5;
      >=I;
      );
      =     "08_LID_MECHANISM_DB".MAGNET_FB_FLT;
      A     L 0.0;
      A     "MAIN_POWER_DB".ALRM_ACK_PB;
      JNB   _00c;
      L     0;
      T     "08_LID_MECHANISM_DB".MAGNET_FB_FLT_TIME;
_00c: NOP   0;
NETWORK
TITLE = LID 1 MAGNET ON COMMAND
      A     "ALWAYS_ON";
      A     "08_LID_MECHANISM_DB".MAGNET_ON_CMD;
      A(;
      A     "08_LID_MECHANISM_DB".LID_INTERLOCK;
      A(;
      A     "08_LID_MECHANISM_DB".LID_MECH_MAN_MD;
      A(;
      O     "08_LID_MECHANISM_DB".MAG_1_STA_PB;
      O     "08_LID_MECHANISM_DB".MAG_1_ON_CMD;
      );
      O;
      A     "08_LID_MECHANISM_DB".LID_MECH_SA_MD;
      A     "08_LID_MECHANISM_DB".PREP_TO_CHRG_SET_BIT;
      A     "08_LID_MECHANISM_DB".LID_1_CAR_FWD_OP_CUT;
      A     "08_LID_MECHANISM_DB".LID_1_VER_DN_OP_CUT;
      AN    "08_LID_MECHANISM_DB".LID_1_VER_DN_CMD_OP_CUT;
      O;
      A     "08_LID_MECHANISM_DB".MAG_1_ON_CMD;
      AN    "08_LID_MECHANISM_DB".LID_1_VER_DN_CMD_OP_CUT;
      );
      O;
      A     "08_LID_MECHANISM_DB".LID_MECH_REP_MD;
      A     "HYDRALIC_DB".HYD_SYS_READY_BIT;
      A(;
      O     "08_LID_MECHANISM_DB".MAG_1_STA_PB;
      O     "08_LID_MECHANISM_DB".MAG_1_ON_CMD;
      );
      );
      A     "08_LID_MECHANISM_DB".MAG_1_STP_PB;
      =     L 0.0;
      A     L 0.0;
      BLD   102;
      =     "08_LID_MECHANISM_DB".MAG_1_ON_CMD;
      A     L 0.0;
      FP    "08_LID_MECHANISM_DB".PULSE_4;
      JNB   _00d;
      L     0;
      T     "08_LID_MECHANISM_DB".LID_1_MAG_ENER_OVER_TIME;
_00d: NOP   0;
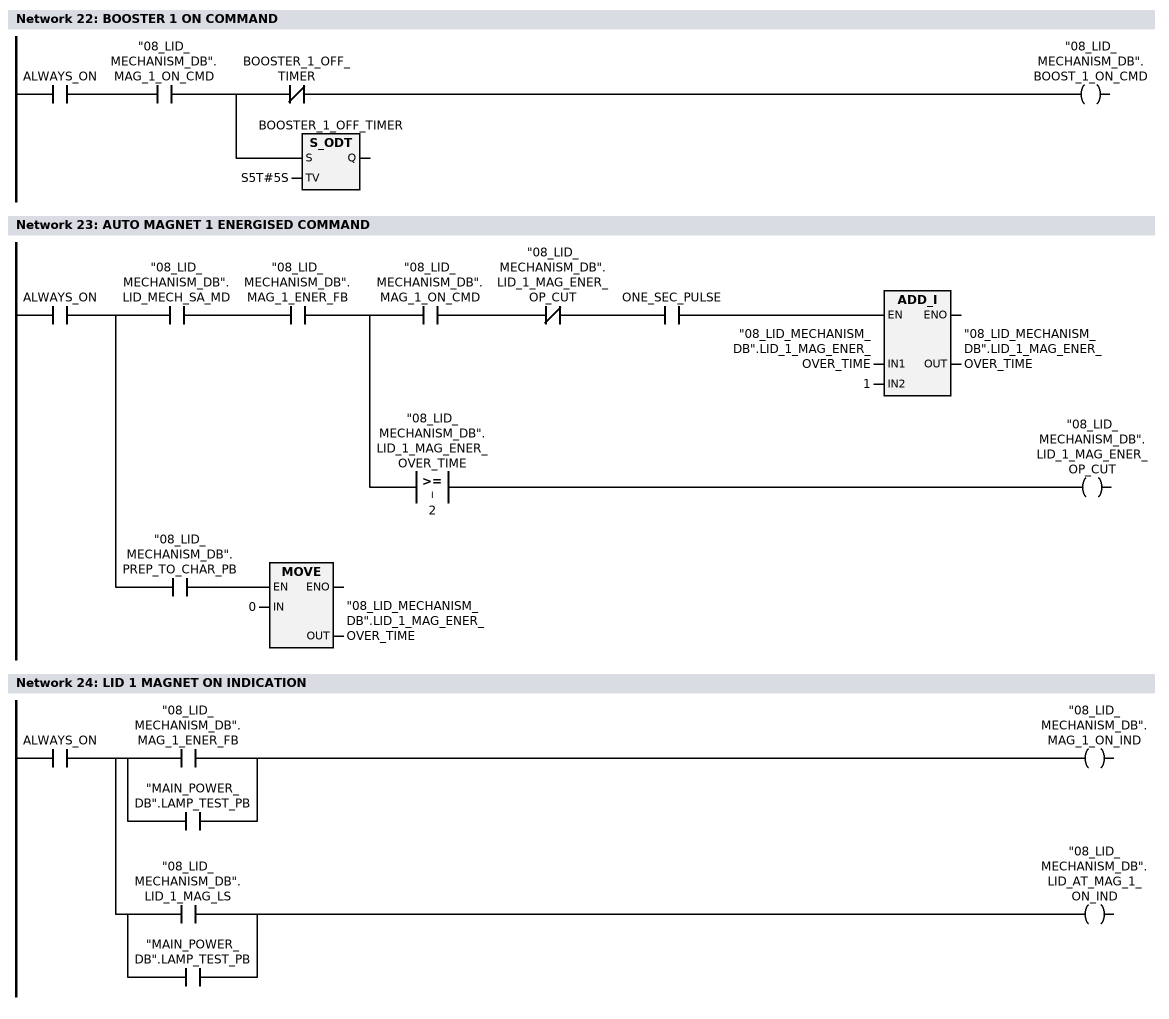
NETWORK
TITLE = BOOSTER 1 ON COMMAND
      A     "ALWAYS_ON";
      A     "08_LID_MECHANISM_DB".MAG_1_ON_CMD;
      =     L 0.0;
      A     L 0.0;
      AN    "BOOSTER_1_OFF_TIMER";
      =     "08_LID_MECHANISM_DB".BOOST_1_ON_CMD;
      A     L 0.0;
      L     S5T#5S;
      SD    "BOOSTER_1_OFF_TIMER";
      NOP   0;
      NOP   0;
      NOP   0;
      NOP   0;
NETWORK
TITLE = AUTO MAGNET 1 ENERGISED COMMAND
      A     "ALWAYS_ON";
      =     L 0.0;
      A     L 0.0;
      A     "08_LID_MECHANISM_DB".LID_MECH_SA_MD;
      A     "08_LID_MECHANISM_DB".MAG_1_ENER_FB;
      =     L 0.1;
      A     L 0.1;
      A     "08_LID_MECHANISM_DB".MAG_1_ON_CMD;
      AN    "08_LID_MECHANISM_DB".LID_1_MAG_ENER_OP_CUT;
      A     "ONE_SEC_PULSE";
      JNB   _00e;
      L     "08_LID_MECHANISM_DB".LID_1_MAG_ENER_OVER_TIME;
      L     1;
      +I;
      T     "08_LID_MECHANISM_DB".LID_1_MAG_ENER_OVER_TIME;
_00e: NOP   0;
      A     L 0.1;
      A(;
      L     "08_LID_MECHANISM_DB".LID_1_MAG_ENER_OVER_TIME;
      L     2;
      >=I;
      );
      =     "08_LID_MECHANISM_DB".LID_1_MAG_ENER_OP_CUT;
      A     L 0.0;
      A     "08_LID_MECHANISM_DB".PREP_TO_CHAR_PB;
      JNB   _00f;
      L     0;
      T     "08_LID_MECHANISM_DB".LID_1_MAG_ENER_OVER_TIME;
_00f: NOP   0;
NETWORK
TITLE = LID 1 MAGNET ON INDICATION
      A     "ALWAYS_ON";
      =     L 0.0;
      A     L 0.0;
      A(;
      O     "08_LID_MECHANISM_DB".MAG_1_ENER_FB;
      O     "MAIN_POWER_DB".LAMP_TEST_PB;
      );
      =     "08_LID_MECHANISM_DB".MAG_1_ON_IND;
      A     L 0.0;
      A(;
      O     "08_LID_MECHANISM_DB".LID_1_MAG_LS;
      O     "MAIN_POWER_DB".LAMP_TEST_PB;
      );
      =     "08_LID_MECHANISM_DB".LID_AT_MAG_1_ON_IND;
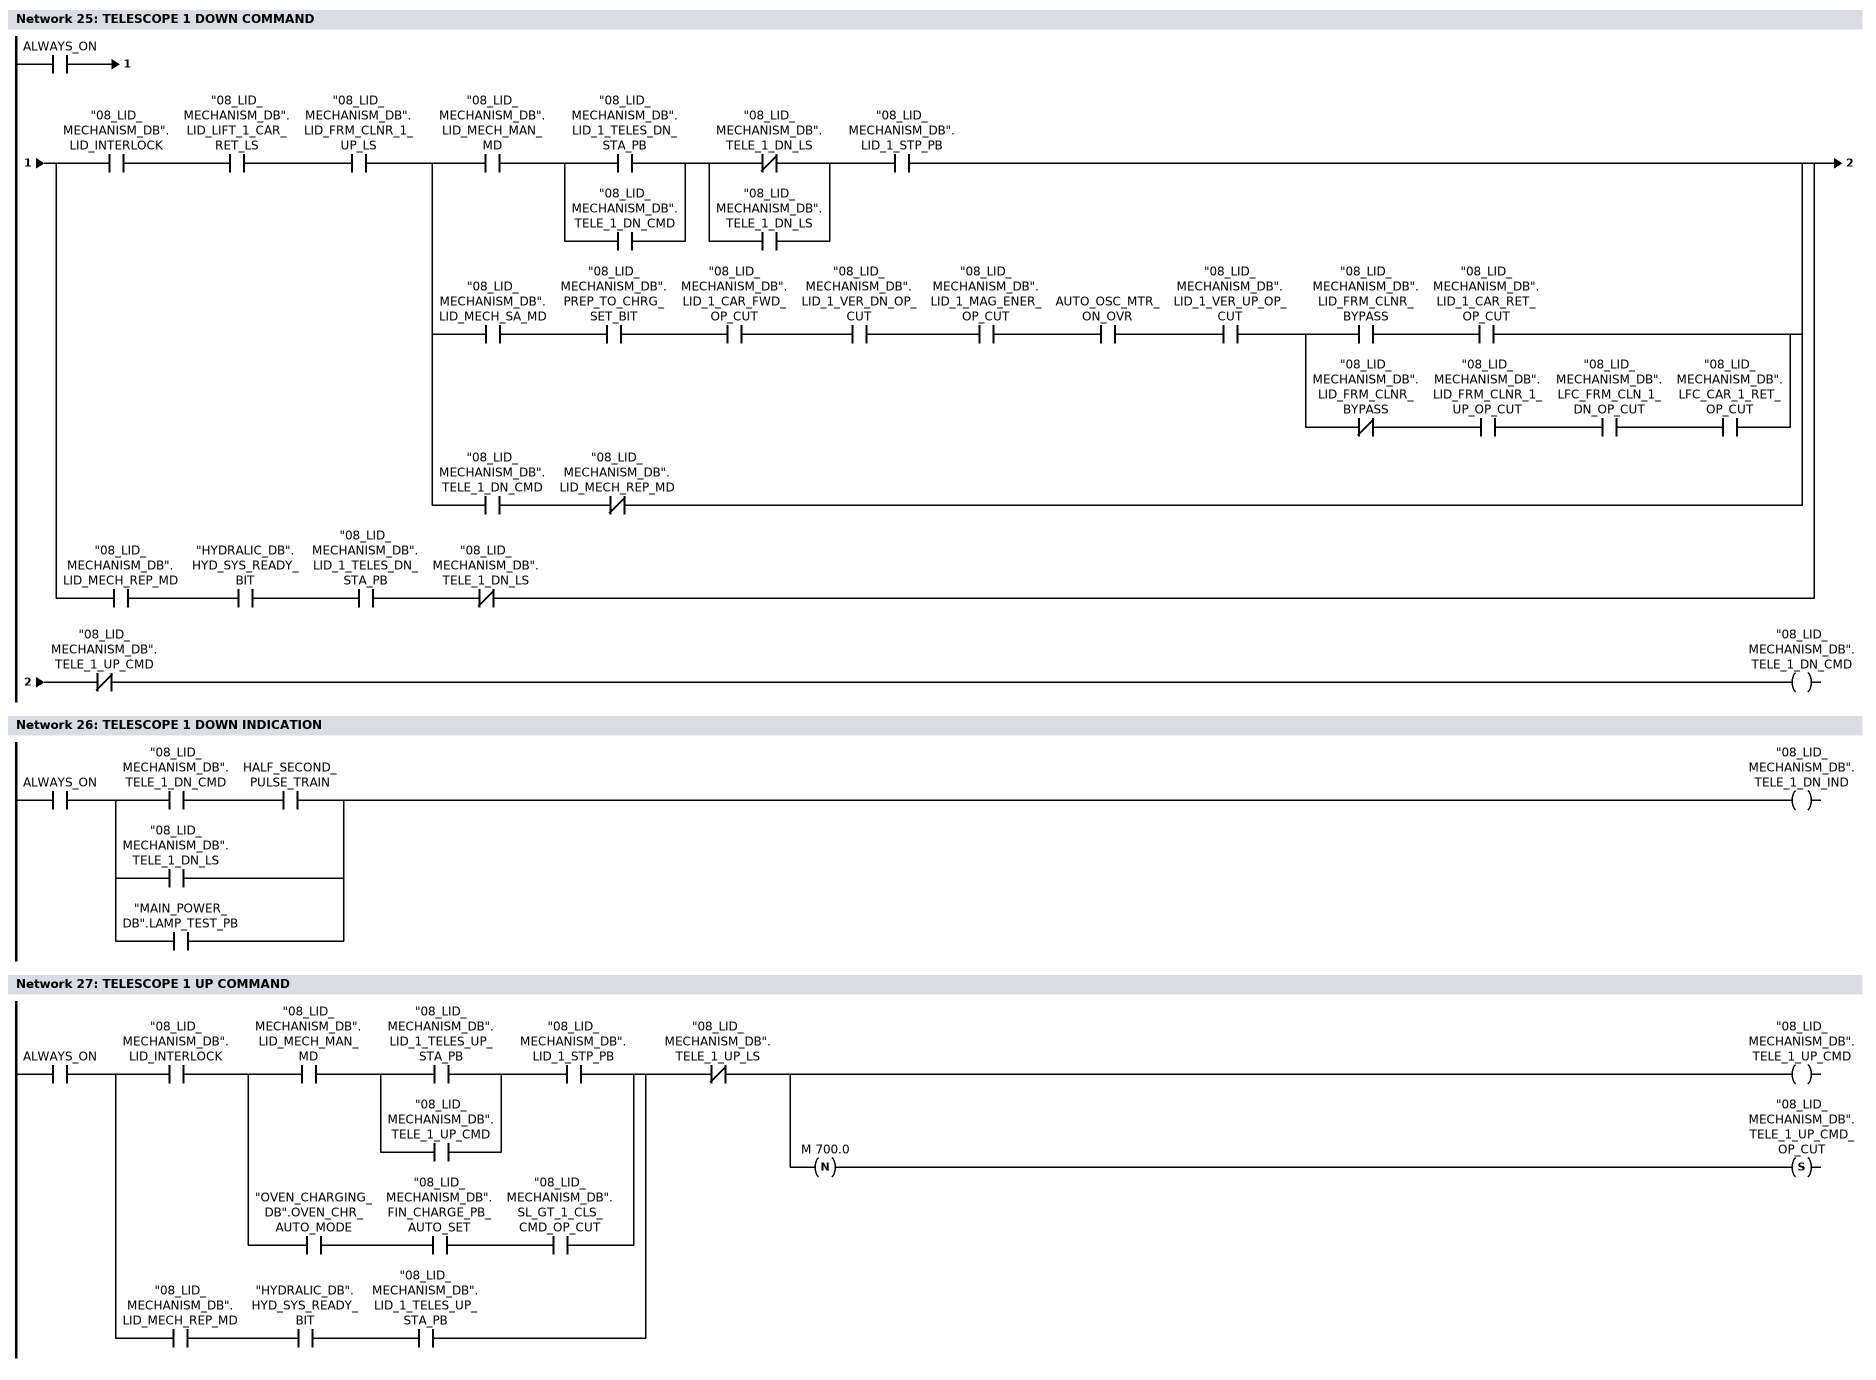
NETWORK
TITLE = TELESCOPE 1 DOWN COMMAND
      A     "ALWAYS_ON";
      A(;
      A     "08_LID_MECHANISM_DB".LID_INTERLOCK;
      A     "08_LID_MECHANISM_DB".LID_LIFT_1_CAR_RET_LS;
      A     "08_LID_MECHANISM_DB".LID_FRM_CLNR_1_UP_LS;
      A(;
      A     "08_LID_MECHANISM_DB".LID_MECH_MAN_MD;
      A(;
      O     "08_LID_MECHANISM_DB".LID_1_TELES_DN_STA_PB;
      O     "08_LID_MECHANISM_DB".TELE_1_DN_CMD;
      );
      A(;
      ON    "08_LID_MECHANISM_DB".TELE_1_DN_LS;
      O     "08_LID_MECHANISM_DB".TELE_1_DN_LS;
      );
      A     "08_LID_MECHANISM_DB".LID_1_STP_PB;
      O;
      A     "08_LID_MECHANISM_DB".LID_MECH_SA_MD;
      A     "08_LID_MECHANISM_DB".PREP_TO_CHRG_SET_BIT;
      A     "08_LID_MECHANISM_DB".LID_1_CAR_FWD_OP_CUT;
      A     "08_LID_MECHANISM_DB".LID_1_VER_DN_OP_CUT;
      A     "08_LID_MECHANISM_DB".LID_1_MAG_ENER_OP_CUT;
      A     "AUTO_OSC_MTR_ON_OVR";
      A     "08_LID_MECHANISM_DB".LID_1_VER_UP_OP_CUT;
      A(;
      A     "08_LID_MECHANISM_DB".LID_FRM_CLNR_BYPASS;
      A     "08_LID_MECHANISM_DB".LID_1_CAR_RET_OP_CUT;
      O;
      AN    "08_LID_MECHANISM_DB".LID_FRM_CLNR_BYPASS;
      A     "08_LID_MECHANISM_DB".LID_FRM_CLNR_1_UP_OP_CUT;
      A     "08_LID_MECHANISM_DB".LFC_FRM_CLN_1_DN_OP_CUT;
      A     "08_LID_MECHANISM_DB".LFC_CAR_1_RET_OP_CUT;
      );
      O;
      A     "08_LID_MECHANISM_DB".TELE_1_DN_CMD;
      AN    "08_LID_MECHANISM_DB".LID_MECH_REP_MD;
      );
      O;
      A     "08_LID_MECHANISM_DB".LID_MECH_REP_MD;
      A     "HYDRALIC_DB".HYD_SYS_READY_BIT;
      A     "08_LID_MECHANISM_DB".LID_1_TELES_DN_STA_PB;
      AN    "08_LID_MECHANISM_DB".TELE_1_DN_LS;
      );
      AN    "08_LID_MECHANISM_DB".TELE_1_UP_CMD;
      =     "08_LID_MECHANISM_DB".TELE_1_DN_CMD;
NETWORK
TITLE = TELESCOPE 1 DOWN INDICATION
      A     "ALWAYS_ON";
      A(;
      A     "08_LID_MECHANISM_DB".TELE_1_DN_CMD;
      A     "HALF_SECOND_PULSE_TRAIN";
      O     "08_LID_MECHANISM_DB".TELE_1_DN_LS;
      O     "MAIN_POWER_DB".LAMP_TEST_PB;
      );
      =     "08_LID_MECHANISM_DB".TELE_1_DN_IND;
NETWORK
TITLE = TELESCOPE 1 UP COMMAND
      A     "ALWAYS_ON";
      A(;
      A     "08_LID_MECHANISM_DB".LID_INTERLOCK;
      A(;
      A     "08_LID_MECHANISM_DB".LID_MECH_MAN_MD;
      A(;
      O     "08_LID_MECHANISM_DB".LID_1_TELES_UP_STA_PB;
      O     "08_LID_MECHANISM_DB".TELE_1_UP_CMD;
      );
      A     "08_LID_MECHANISM_DB".LID_1_STP_PB;
      O;
      A     "OVEN_CHARGING_DB".OVEN_CHR_AUTO_MODE;
      A     "08_LID_MECHANISM_DB".FIN_CHARGE_PB_AUTO_SET;
      A     "08_LID_MECHANISM_DB".SL_GT_1_CLS_CMD_OP_CUT;
      );
      O;
      A     "08_LID_MECHANISM_DB".LID_MECH_REP_MD;
      A     "HYDRALIC_DB".HYD_SYS_READY_BIT;
      A     "08_LID_MECHANISM_DB".LID_1_TELES_UP_STA_PB;
      );
      AN    "08_LID_MECHANISM_DB".TELE_1_UP_LS;
      =     L 0.0;
      A     L 0.0;
      BLD   102;
      =     "08_LID_MECHANISM_DB".TELE_1_UP_CMD;
      A     L 0.0;
      FN    M 700.0;
      S     "08_LID_MECHANISM_DB".TELE_1_UP_CMD_OP_CUT;
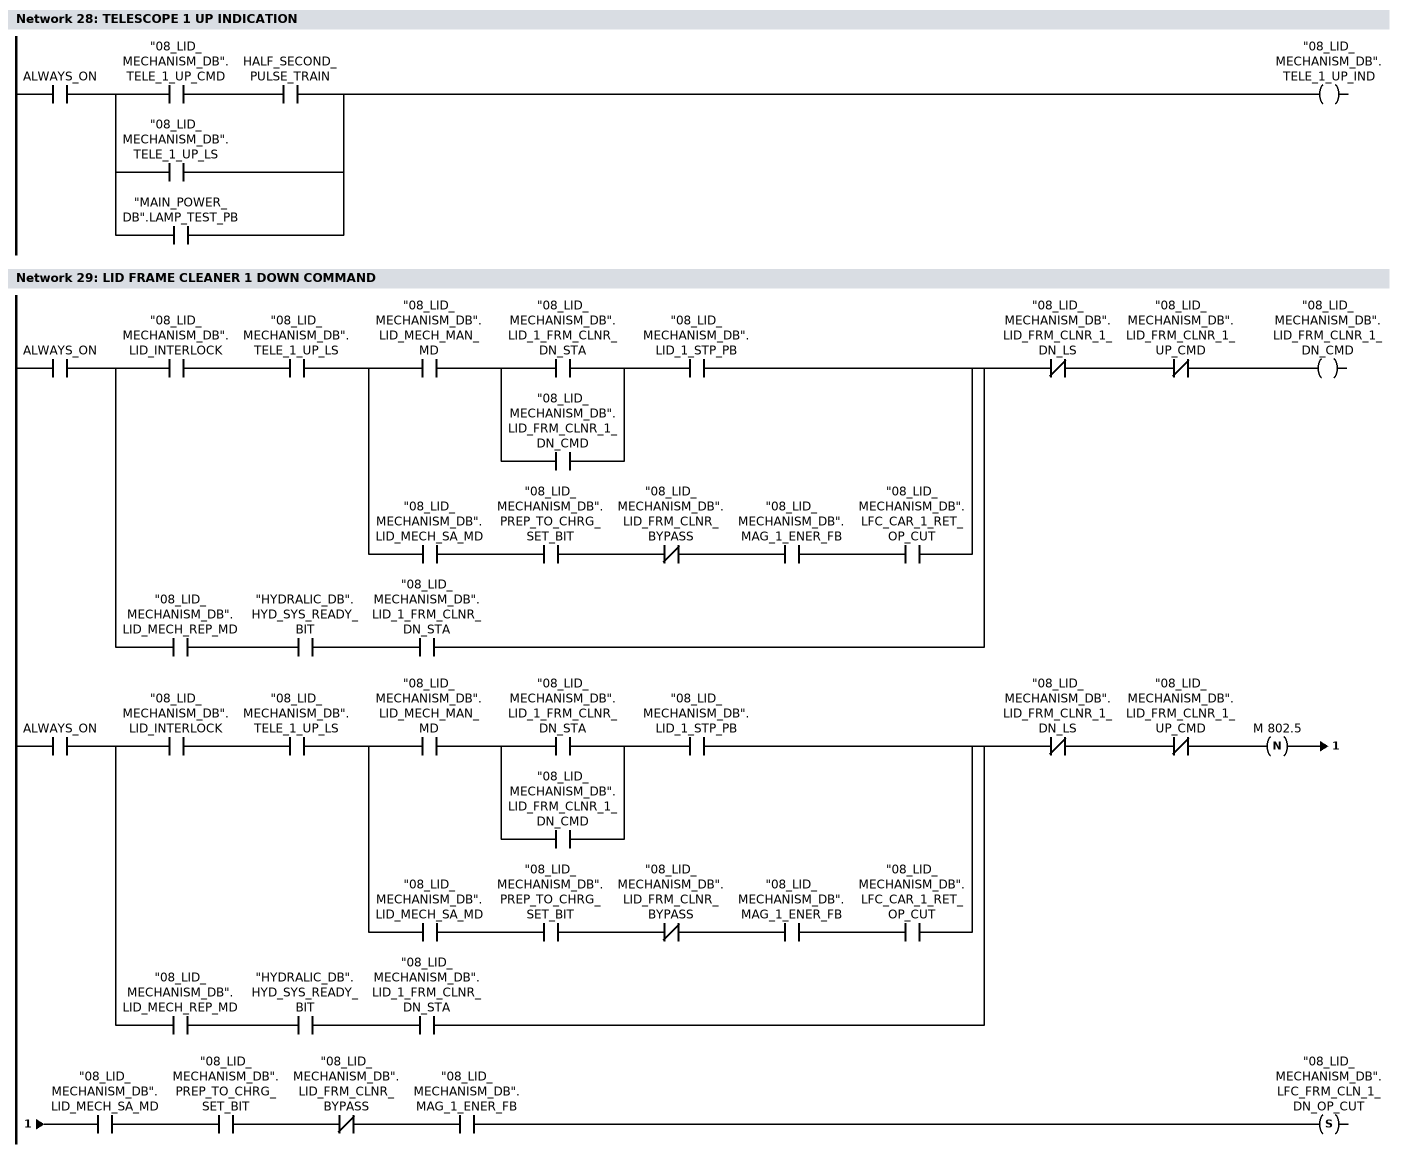
NETWORK
TITLE = TELESCOPE 1 UP INDICATION
      A     "ALWAYS_ON";
      A(;
      A     "08_LID_MECHANISM_DB".TELE_1_UP_CMD;
      A     "HALF_SECOND_PULSE_TRAIN";
      O     "08_LID_MECHANISM_DB".TELE_1_UP_LS;
      O     "MAIN_POWER_DB".LAMP_TEST_PB;
      );
      =     "08_LID_MECHANISM_DB".TELE_1_UP_IND;
NETWORK
TITLE = LID FRAME CLEANER 1 DOWN COMMAND
      A     "ALWAYS_ON";
      A(;
      A     "08_LID_MECHANISM_DB".LID_INTERLOCK;
      A     "08_LID_MECHANISM_DB".TELE_1_UP_LS;
      A(;
      A     "08_LID_MECHANISM_DB".LID_MECH_MAN_MD;
      A(;
      O     "08_LID_MECHANISM_DB".LID_1_FRM_CLNR_DN_STA;
      O     "08_LID_MECHANISM_DB".LID_FRM_CLNR_1_DN_CMD;
      );
      A     "08_LID_MECHANISM_DB".LID_1_STP_PB;
      O;
      A     "08_LID_MECHANISM_DB".LID_MECH_SA_MD;
      A     "08_LID_MECHANISM_DB".PREP_TO_CHRG_SET_BIT;
      AN    "08_LID_MECHANISM_DB".LID_FRM_CLNR_BYPASS;
      A     "08_LID_MECHANISM_DB".MAG_1_ENER_FB;
      A     "08_LID_MECHANISM_DB".LFC_CAR_1_RET_OP_CUT;
      );
      O;
      A     "08_LID_MECHANISM_DB".LID_MECH_REP_MD;
      A     "HYDRALIC_DB".HYD_SYS_READY_BIT;
      A     "08_LID_MECHANISM_DB".LID_1_FRM_CLNR_DN_STA;
      );
      AN    "08_LID_MECHANISM_DB".LID_FRM_CLNR_1_DN_LS;
      AN    "08_LID_MECHANISM_DB".LID_FRM_CLNR_1_UP_CMD;
      =     L 0.0;
      A     L 0.0;
      BLD   102;
      =     "08_LID_MECHANISM_DB".LID_FRM_CLNR_1_DN_CMD;
      A(;
      A     L 0.0;
      FN    M 802.5;
      );
      A     "08_LID_MECHANISM_DB".LID_MECH_SA_MD;
      A     "08_LID_MECHANISM_DB".PREP_TO_CHRG_SET_BIT;
      AN    "08_LID_MECHANISM_DB".LID_FRM_CLNR_BYPASS;
      A     "08_LID_MECHANISM_DB".MAG_1_ENER_FB;
      S     "08_LID_MECHANISM_DB".LFC_FRM_CLN_1_DN_OP_CUT;
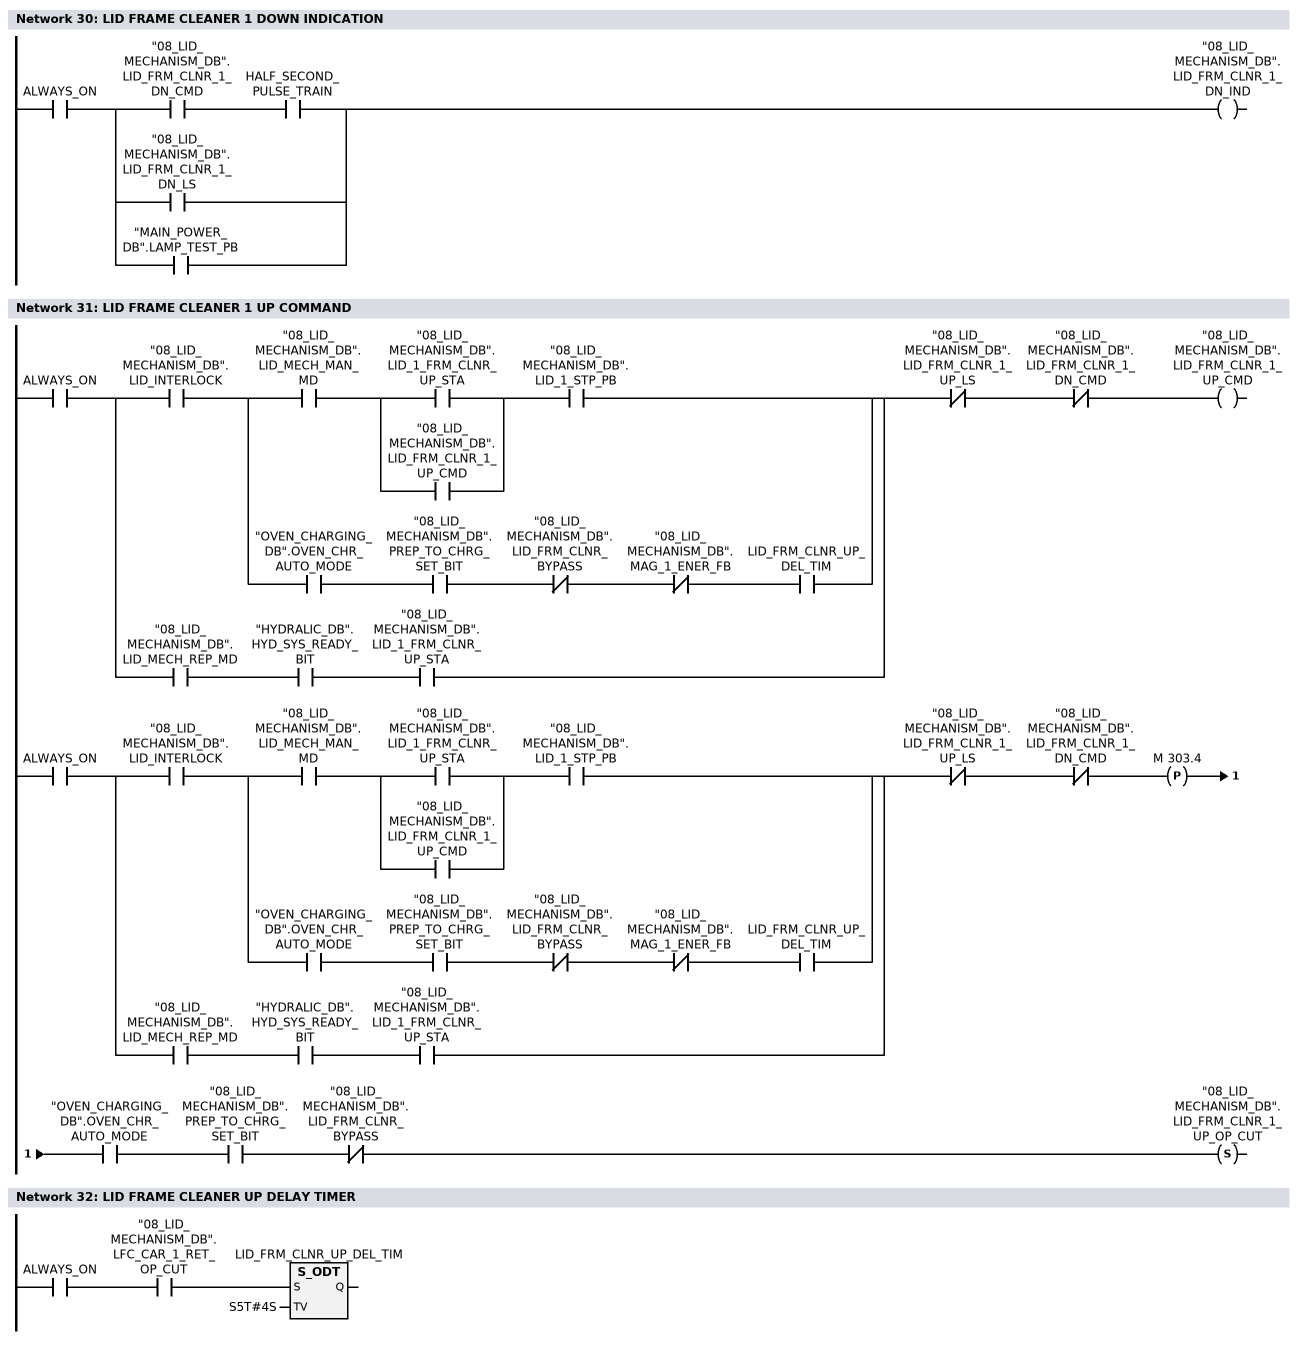
NETWORK
TITLE = LID FRAME CLEANER 1 DOWN INDICATION
      A     "ALWAYS_ON";
      A(;
      A     "08_LID_MECHANISM_DB".LID_FRM_CLNR_1_DN_CMD;
      A     "HALF_SECOND_PULSE_TRAIN";
      O     "08_LID_MECHANISM_DB".LID_FRM_CLNR_1_DN_LS;
      O     "MAIN_POWER_DB".LAMP_TEST_PB;
      );
      =     "08_LID_MECHANISM_DB".LID_FRM_CLNR_1_DN_IND;
NETWORK
TITLE = LID FRAME CLEANER 1 UP COMMAND
      A     "ALWAYS_ON";
      A(;
      A     "08_LID_MECHANISM_DB".LID_INTERLOCK;
      A(;
      A     "08_LID_MECHANISM_DB".LID_MECH_MAN_MD;
      A(;
      O     "08_LID_MECHANISM_DB".LID_1_FRM_CLNR_UP_STA;
      O     "08_LID_MECHANISM_DB".LID_FRM_CLNR_1_UP_CMD;
      );
      A     "08_LID_MECHANISM_DB".LID_1_STP_PB;
      O;
      A     "OVEN_CHARGING_DB".OVEN_CHR_AUTO_MODE;
      A     "08_LID_MECHANISM_DB".PREP_TO_CHRG_SET_BIT;
      AN    "08_LID_MECHANISM_DB".LID_FRM_CLNR_BYPASS;
      AN    "08_LID_MECHANISM_DB".MAG_1_ENER_FB;
      A     "LID_FRM_CLNR_UP_DEL_TIM";
      );
      O;
      A     "08_LID_MECHANISM_DB".LID_MECH_REP_MD;
      A     "HYDRALIC_DB".HYD_SYS_READY_BIT;
      A     "08_LID_MECHANISM_DB".LID_1_FRM_CLNR_UP_STA;
      );
      AN    "08_LID_MECHANISM_DB".LID_FRM_CLNR_1_UP_LS;
      AN    "08_LID_MECHANISM_DB".LID_FRM_CLNR_1_DN_CMD;
      =     L 0.0;
      A     L 0.0;
      BLD   102;
      =     "08_LID_MECHANISM_DB".LID_FRM_CLNR_1_UP_CMD;
      A(;
      A     L 0.0;
      FP    M 303.4;
      );
      A     "OVEN_CHARGING_DB".OVEN_CHR_AUTO_MODE;
      A     "08_LID_MECHANISM_DB".PREP_TO_CHRG_SET_BIT;
      AN    "08_LID_MECHANISM_DB".LID_FRM_CLNR_BYPASS;
      S     "08_LID_MECHANISM_DB".LID_FRM_CLNR_1_UP_OP_CUT;
NETWORK
TITLE = LID FRAME CLEANER UP DELAY TIMER
      A     "ALWAYS_ON";
      A     "08_LID_MECHANISM_DB".LFC_CAR_1_RET_OP_CUT;
      L     S5T#4S;
      SD    "LID_FRM_CLNR_UP_DEL_TIM";
      NOP   0;
      NOP   0;
      NOP   0;
      NOP   0;
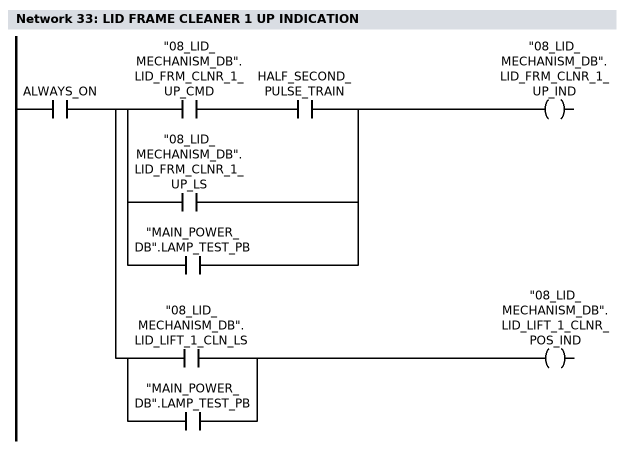
NETWORK
TITLE = LID FRAME CLEANER 1 UP INDICATION
      A     "ALWAYS_ON";
      =     L 0.0;
      A     L 0.0;
      A(;
      A     "08_LID_MECHANISM_DB".LID_FRM_CLNR_1_UP_CMD;
      A     "HALF_SECOND_PULSE_TRAIN";
      O     "08_LID_MECHANISM_DB".LID_FRM_CLNR_1_UP_LS;
      O     "MAIN_POWER_DB".LAMP_TEST_PB;
      );
      =     "08_LID_MECHANISM_DB".LID_FRM_CLNR_1_UP_IND;
      A     L 0.0;
      A(;
      O     "08_LID_MECHANISM_DB".LID_LIFT_1_CLN_LS;
      O     "MAIN_POWER_DB".LAMP_TEST_PB;
      );
      =     "08_LID_MECHANISM_DB".LID_LIFT_1_CLNR_POS_IND;
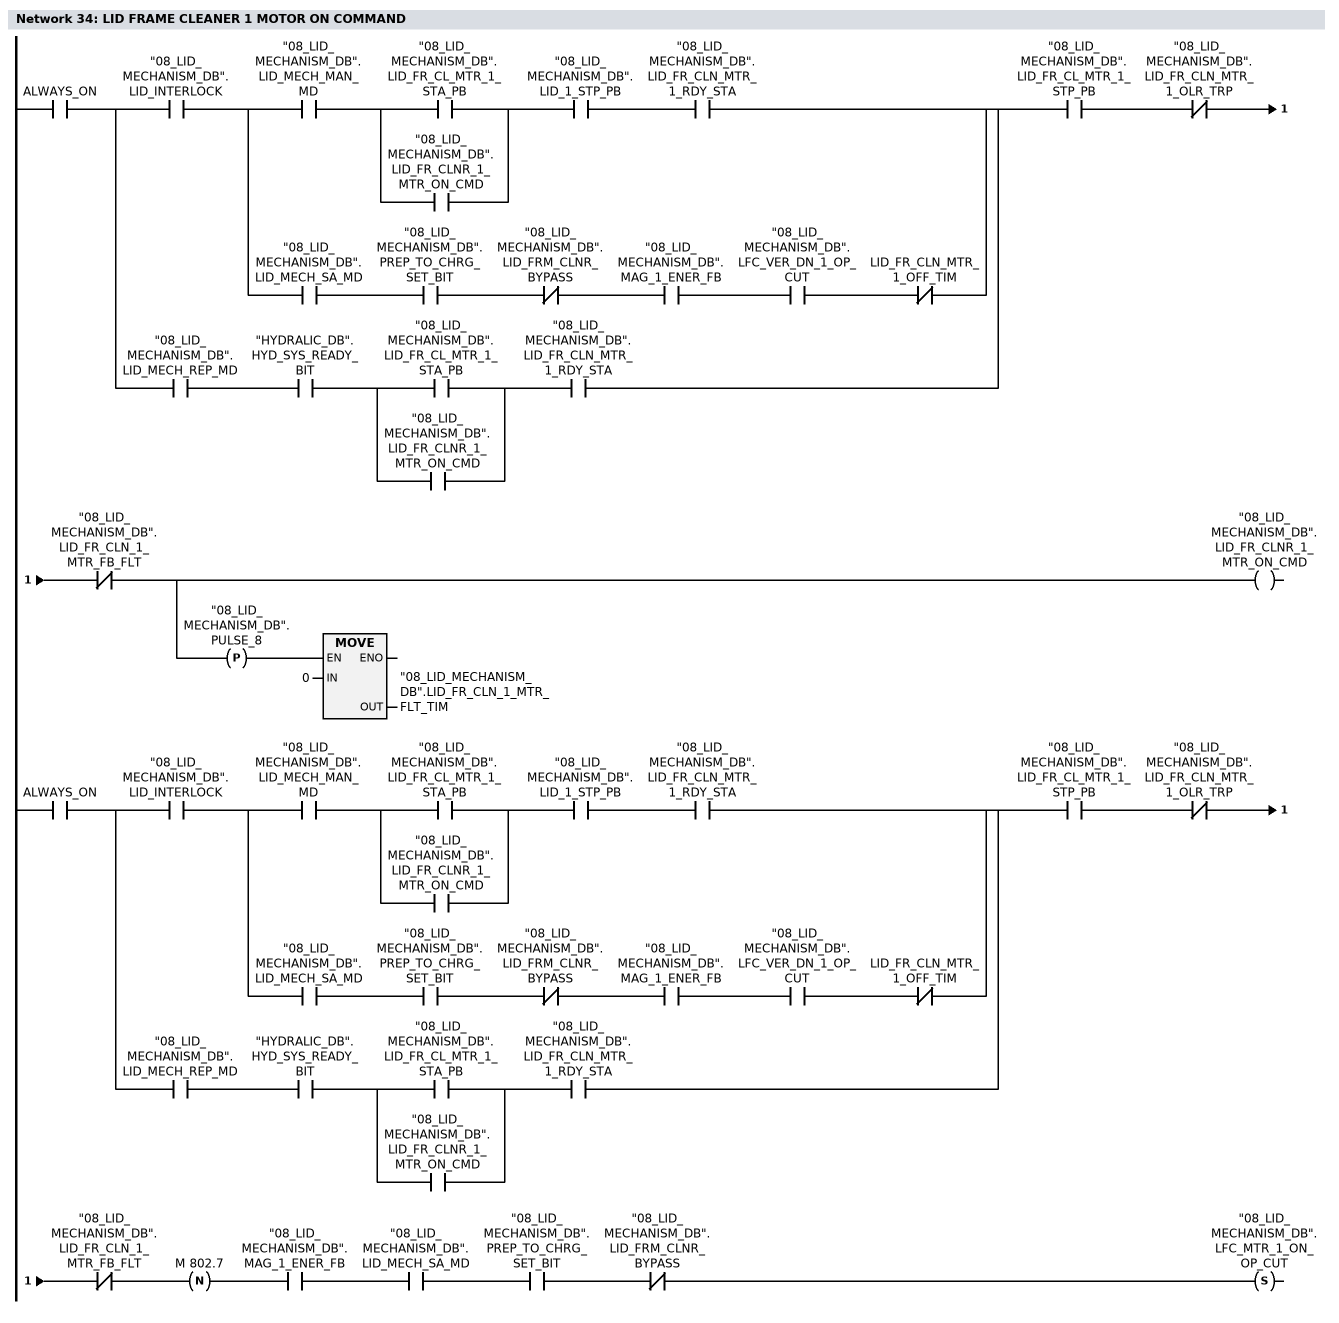
NETWORK
TITLE = LID FRAME CLEANER 1 MOTOR ON COMMAND
      A     "ALWAYS_ON";
      A(;
      A     "08_LID_MECHANISM_DB".LID_INTERLOCK;
      A(;
      A     "08_LID_MECHANISM_DB".LID_MECH_MAN_MD;
      A(;
      O     "08_LID_MECHANISM_DB".LID_FR_CL_MTR_1_STA_PB;
      O     "08_LID_MECHANISM_DB".LID_FR_CLNR_1_MTR_ON_CMD;
      );
      A     "08_LID_MECHANISM_DB".LID_1_STP_PB;
      A     "08_LID_MECHANISM_DB".LID_FR_CLN_MTR_1_RDY_STA;
      O;
      A     "08_LID_MECHANISM_DB".LID_MECH_SA_MD;
      A     "08_LID_MECHANISM_DB".PREP_TO_CHRG_SET_BIT;
      AN    "08_LID_MECHANISM_DB".LID_FRM_CLNR_BYPASS;
      A     "08_LID_MECHANISM_DB".MAG_1_ENER_FB;
      A     "08_LID_MECHANISM_DB".LFC_VER_DN_1_OP_CUT;
      AN    "LID_FR_CLN_MTR_1_OFF_TIM";
      );
      O;
      A     "08_LID_MECHANISM_DB".LID_MECH_REP_MD;
      A     "HYDRALIC_DB".HYD_SYS_READY_BIT;
      A(;
      O     "08_LID_MECHANISM_DB".LID_FR_CL_MTR_1_STA_PB;
      O     "08_LID_MECHANISM_DB".LID_FR_CLNR_1_MTR_ON_CMD;
      );
      A     "08_LID_MECHANISM_DB".LID_FR_CLN_MTR_1_RDY_STA;
      );
      A     "08_LID_MECHANISM_DB".LID_FR_CL_MTR_1_STP_PB;
      AN    "08_LID_MECHANISM_DB".LID_FR_CLN_MTR_1_OLR_TRP;
      AN    "08_LID_MECHANISM_DB".LID_FR_CLN_1_MTR_FB_FLT;
      =     L 0.0;
      A     L 0.0;
      BLD   102;
      =     "08_LID_MECHANISM_DB".LID_FR_CLNR_1_MTR_ON_CMD;
      A     L 0.0;
      FP    "08_LID_MECHANISM_DB".PULSE_8;
      JNB   _010;
      L     0;
      T     "08_LID_MECHANISM_DB".LID_FR_CLN_1_MTR_FLT_TIM;
_010: NOP   0;
      A(;
      A     L 0.0;
      FN    M 802.7;
      );
      A     "08_LID_MECHANISM_DB".MAG_1_ENER_FB;
      A     "08_LID_MECHANISM_DB".LID_MECH_SA_MD;
      A     "08_LID_MECHANISM_DB".PREP_TO_CHRG_SET_BIT;
      AN    "08_LID_MECHANISM_DB".LID_FRM_CLNR_BYPASS;
      S     "08_LID_MECHANISM_DB".LFC_MTR_1_ON_OP_CUT;
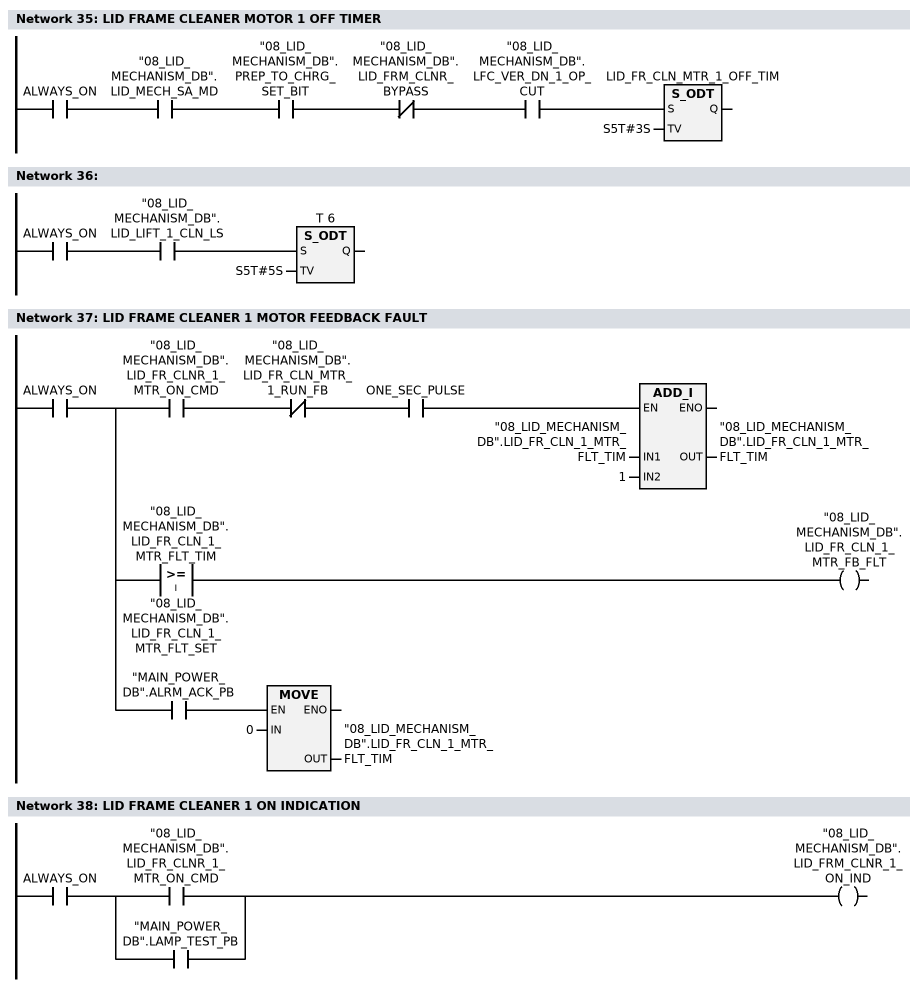
NETWORK
TITLE = LID FRAME CLEANER MOTOR 1 OFF TIMER
      A     "ALWAYS_ON";
      A     "08_LID_MECHANISM_DB".LID_MECH_SA_MD;
      A     "08_LID_MECHANISM_DB".PREP_TO_CHRG_SET_BIT;
      AN    "08_LID_MECHANISM_DB".LID_FRM_CLNR_BYPASS;
      A     "08_LID_MECHANISM_DB".LFC_VER_DN_1_OP_CUT;
      L     S5T#3S;
      SD    "LID_FR_CLN_MTR_1_OFF_TIM";
      NOP   0;
      NOP   0;
      NOP   0;
      NOP   0;
NETWORK
TITLE =
      A     "ALWAYS_ON";
      A     "08_LID_MECHANISM_DB".LID_LIFT_1_CLN_LS;
      L     S5T#5S;
      SD    T 6;
      NOP   0;
      NOP   0;
      NOP   0;
      NOP   0;
NETWORK
TITLE = LID FRAME CLEANER 1 MOTOR FEEDBACK FAULT
      A     "ALWAYS_ON";
      =     L 0.0;
      A     L 0.0;
      A     "08_LID_MECHANISM_DB".LID_FR_CLNR_1_MTR_ON_CMD;
      AN    "08_LID_MECHANISM_DB".LID_FR_CLN_MTR_1_RUN_FB;
      A     "ONE_SEC_PULSE";
      JNB   _011;
      L     "08_LID_MECHANISM_DB".LID_FR_CLN_1_MTR_FLT_TIM;
      L     1;
      +I;
      T     "08_LID_MECHANISM_DB".LID_FR_CLN_1_MTR_FLT_TIM;
_011: NOP   0;
      A     L 0.0;
      A(;
      L     "08_LID_MECHANISM_DB".LID_FR_CLN_1_MTR_FLT_TIM;
      L     "08_LID_MECHANISM_DB".LID_FR_CLN_1_MTR_FLT_SET;
      >=I;
      );
      =     "08_LID_MECHANISM_DB".LID_FR_CLN_1_MTR_FB_FLT;
      A     L 0.0;
      A     "MAIN_POWER_DB".ALRM_ACK_PB;
      JNB   _012;
      L     0;
      T     "08_LID_MECHANISM_DB".LID_FR_CLN_1_MTR_FLT_TIM;
_012: NOP   0;
NETWORK
TITLE = LID FRAME CLEANER 1 ON INDICATION
      A     "ALWAYS_ON";
      A(;
      O     "08_LID_MECHANISM_DB".LID_FR_CLNR_1_MTR_ON_CMD;
      O     "MAIN_POWER_DB".LAMP_TEST_PB;
      );
      =     "08_LID_MECHANISM_DB".LID_FRM_CLNR_1_ON_IND;
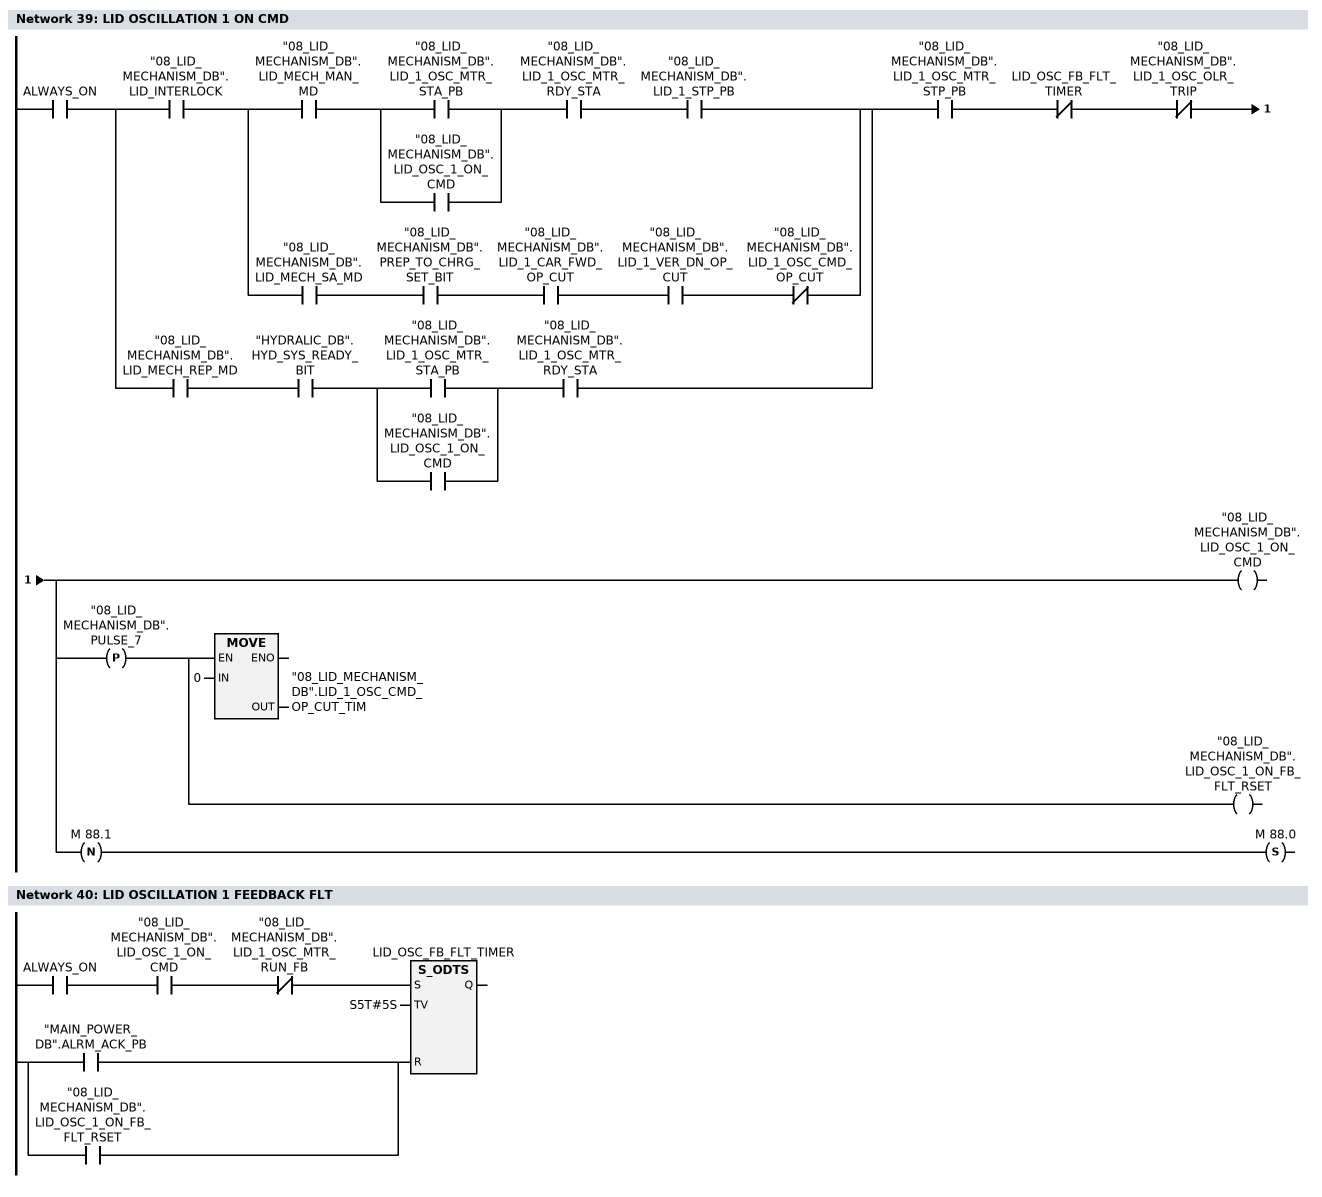
NETWORK
TITLE = LID OSCILLATION 1 ON CMD
      A     "ALWAYS_ON";
      A(;
      A     "08_LID_MECHANISM_DB".LID_INTERLOCK;
      A(;
      A     "08_LID_MECHANISM_DB".LID_MECH_MAN_MD;
      A(;
      O     "08_LID_MECHANISM_DB".LID_1_OSC_MTR_STA_PB;
      O     "08_LID_MECHANISM_DB".LID_OSC_1_ON_CMD;
      );
      A     "08_LID_MECHANISM_DB".LID_1_OSC_MTR_RDY_STA;
      A     "08_LID_MECHANISM_DB".LID_1_STP_PB;
      O;
      A     "08_LID_MECHANISM_DB".LID_MECH_SA_MD;
      A     "08_LID_MECHANISM_DB".PREP_TO_CHRG_SET_BIT;
      A     "08_LID_MECHANISM_DB".LID_1_CAR_FWD_OP_CUT;
      A     "08_LID_MECHANISM_DB".LID_1_VER_DN_OP_CUT;
      AN    "08_LID_MECHANISM_DB".LID_1_OSC_CMD_OP_CUT;
      );
      O;
      A     "08_LID_MECHANISM_DB".LID_MECH_REP_MD;
      A     "HYDRALIC_DB".HYD_SYS_READY_BIT;
      A(;
      O     "08_LID_MECHANISM_DB".LID_1_OSC_MTR_STA_PB;
      O     "08_LID_MECHANISM_DB".LID_OSC_1_ON_CMD;
      );
      A     "08_LID_MECHANISM_DB".LID_1_OSC_MTR_RDY_STA;
      );
      A     "08_LID_MECHANISM_DB".LID_1_OSC_MTR_STP_PB;
      AN    "LID_OSC_FB_FLT_TIMER";
      AN    "08_LID_MECHANISM_DB".LID_1_OSC_OLR_TRIP;
      =     L 0.0;
      A     L 0.0;
      BLD   102;
      =     "08_LID_MECHANISM_DB".LID_OSC_1_ON_CMD;
      A     L 0.0;
      FP    "08_LID_MECHANISM_DB".PULSE_7;
      =     L 0.1;
      A     L 0.1;
      JNB   _013;
      L     0;
      T     "08_LID_MECHANISM_DB".LID_1_OSC_CMD_OP_CUT_TIM;
_013: NOP   0;
      A     L 0.1;
      BLD   102;
      =     "08_LID_MECHANISM_DB".LID_OSC_1_ON_FB_FLT_RSET;
      A     L 0.0;
      FN    M 88.1;
      S     M 88.0;
NETWORK
TITLE = LID OSCILLATION 1 FEEDBACK FLT
      A     "ALWAYS_ON";
      A     "08_LID_MECHANISM_DB".LID_OSC_1_ON_CMD;
      AN    "08_LID_MECHANISM_DB".LID_1_OSC_MTR_RUN_FB;
      L     S5T#5S;
      SS    "LID_OSC_FB_FLT_TIMER";
      A(;
      O     "MAIN_POWER_DB".ALRM_ACK_PB;
      O     "08_LID_MECHANISM_DB".LID_OSC_1_ON_FB_FLT_RSET;
      );
      R     "LID_OSC_FB_FLT_TIMER";
      NOP   0;
      NOP   0;
      NOP   0;
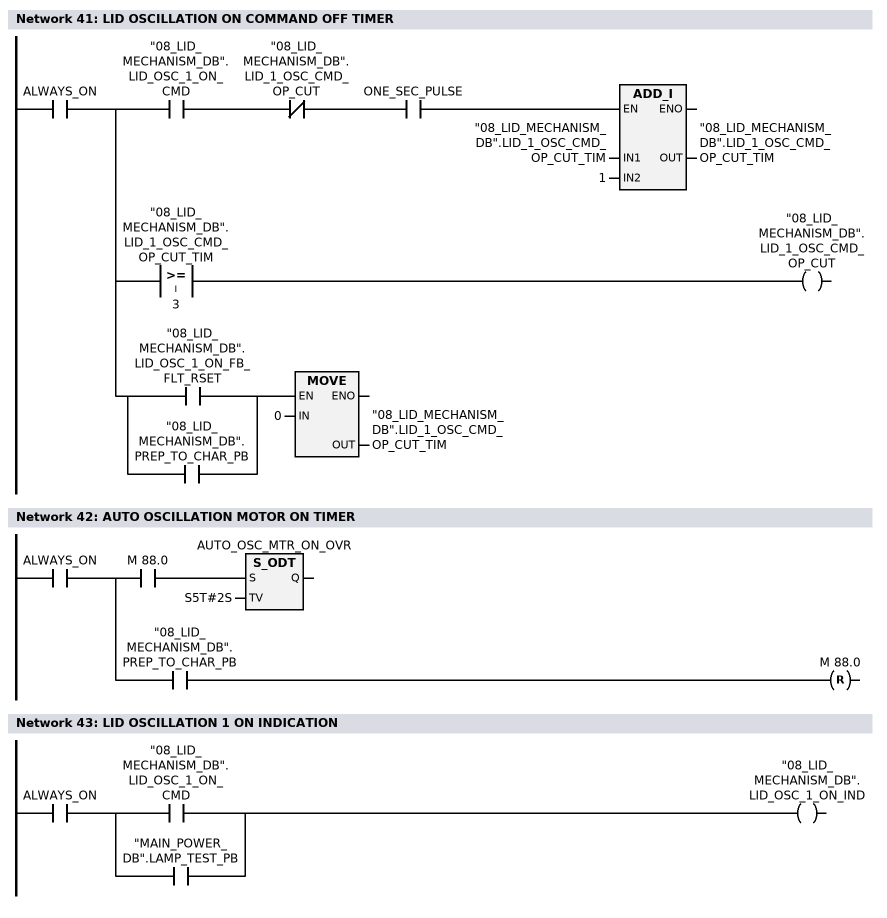
NETWORK
TITLE = LID OSCILLATION ON COMMAND OFF TIMER
      A     "ALWAYS_ON";
      =     L 0.0;
      A     L 0.0;
      A     "08_LID_MECHANISM_DB".LID_OSC_1_ON_CMD;
      AN    "08_LID_MECHANISM_DB".LID_1_OSC_CMD_OP_CUT;
      A     "ONE_SEC_PULSE";
      JNB   _014;
      L     "08_LID_MECHANISM_DB".LID_1_OSC_CMD_OP_CUT_TIM;
      L     1;
      +I;
      T     "08_LID_MECHANISM_DB".LID_1_OSC_CMD_OP_CUT_TIM;
_014: NOP   0;
      A     L 0.0;
      A(;
      L     "08_LID_MECHANISM_DB".LID_1_OSC_CMD_OP_CUT_TIM;
      L     3;
      >=I;
      );
      =     "08_LID_MECHANISM_DB".LID_1_OSC_CMD_OP_CUT;
      A     L 0.0;
      A(;
      O     "08_LID_MECHANISM_DB".LID_OSC_1_ON_FB_FLT_RSET;
      O     "08_LID_MECHANISM_DB".PREP_TO_CHAR_PB;
      );
      JNB   _015;
      L     0;
      T     "08_LID_MECHANISM_DB".LID_1_OSC_CMD_OP_CUT_TIM;
_015: NOP   0;
NETWORK
TITLE = AUTO OSCILLATION MOTOR ON TIMER
      A     "ALWAYS_ON";
      =     L 0.0;
      A     L 0.0;
      A     M 88.0;
      L     S5T#2S;
      SD    "AUTO_OSC_MTR_ON_OVR";
      NOP   0;
      NOP   0;
      NOP   0;
      NOP   0;
      A     L 0.0;
      A     "08_LID_MECHANISM_DB".PREP_TO_CHAR_PB;
      R     M 88.0;
NETWORK
TITLE = LID OSCILLATION 1 ON INDICATION
      A     "ALWAYS_ON";
      A(;
      O     "08_LID_MECHANISM_DB".LID_OSC_1_ON_CMD;
      O     "MAIN_POWER_DB".LAMP_TEST_PB;
      );
      =     "08_LID_MECHANISM_DB".LID_OSC_1_ON_IND;
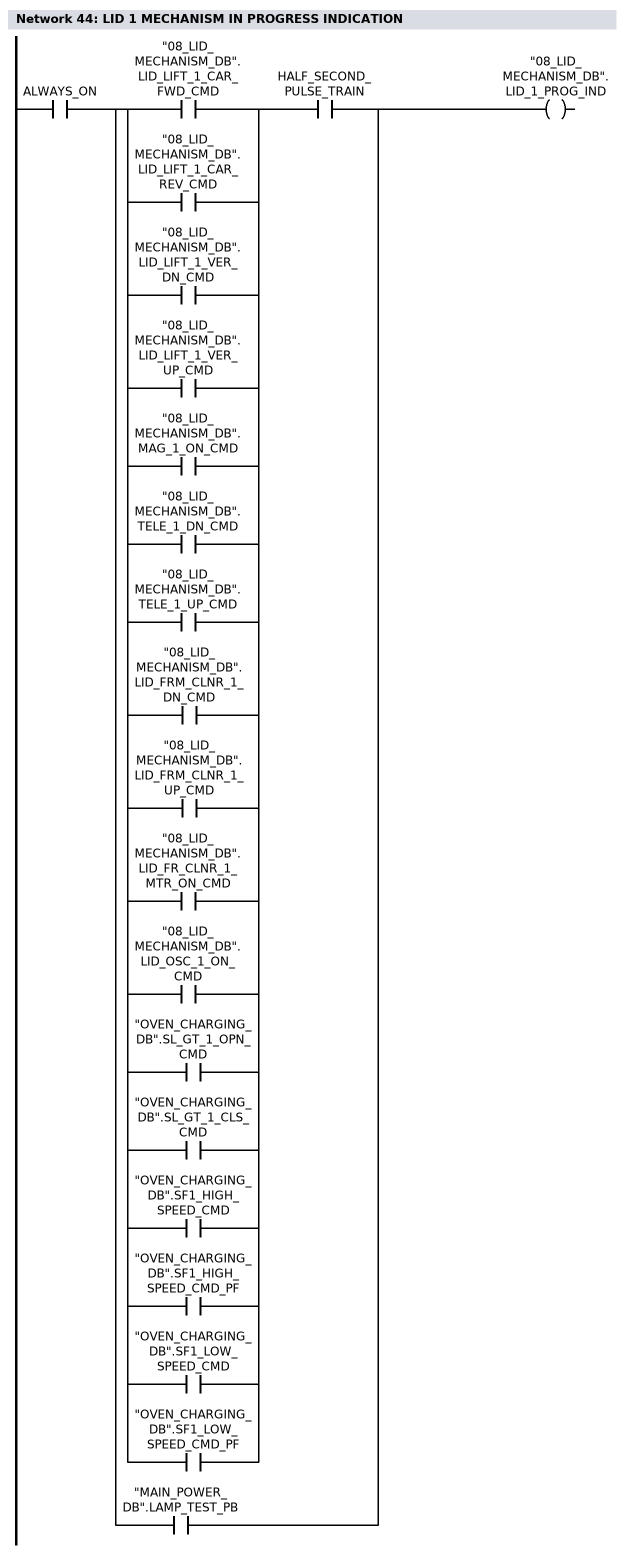
NETWORK
TITLE = LID 1 MECHANISM IN PROGRESS INDICATION
      A     "ALWAYS_ON";
      A(;
      A(;
      O     "08_LID_MECHANISM_DB".LID_LIFT_1_CAR_FWD_CMD;
      O     "08_LID_MECHANISM_DB".LID_LIFT_1_CAR_REV_CMD;
      O     "08_LID_MECHANISM_DB".LID_LIFT_1_VER_DN_CMD;
      O     "08_LID_MECHANISM_DB".LID_LIFT_1_VER_UP_CMD;
      O     "08_LID_MECHANISM_DB".MAG_1_ON_CMD;
      O     "08_LID_MECHANISM_DB".TELE_1_DN_CMD;
      O     "08_LID_MECHANISM_DB".TELE_1_UP_CMD;
      O     "08_LID_MECHANISM_DB".LID_FRM_CLNR_1_DN_CMD;
      O     "08_LID_MECHANISM_DB".LID_FRM_CLNR_1_UP_CMD;
      O     "08_LID_MECHANISM_DB".LID_FR_CLNR_1_MTR_ON_CMD;
      O     "08_LID_MECHANISM_DB".LID_OSC_1_ON_CMD;
      O     "OVEN_CHARGING_DB".SL_GT_1_OPN_CMD;
      O     "OVEN_CHARGING_DB".SL_GT_1_CLS_CMD;
      O     "OVEN_CHARGING_DB".SF1_HIGH_SPEED_CMD;
      O     "OVEN_CHARGING_DB".SF1_HIGH_SPEED_CMD_PF;
      O     "OVEN_CHARGING_DB".SF1_LOW_SPEED_CMD;
      O     "OVEN_CHARGING_DB".SF1_LOW_SPEED_CMD_PF;
      );
      A     "HALF_SECOND_PULSE_TRAIN";
      O     "MAIN_POWER_DB".LAMP_TEST_PB;
      );
      =     "08_LID_MECHANISM_DB".LID_1_PROG_IND;
END_FUNCTION

FUNCTION "PROFIBUS COMMUNICATION" : VOID	// FC 12
AUTHOR : Arun_Ram
VERSION : 0.1
VAR_TEMP
  TEMP1 : INT ;
  TEMP2 : INT ;
  TEMP3 : INT ;
  TEMP4 : INT ;
  TEMP5 : INT ;
  TEMP6 : INT ;
  TEMP7 : INT ;
  TEMP8 : INT ;
  TEMP9 : WORD ;
  TEMP10 : INT ;
  TEMP11 : INT ;
  TEMP12 : INT ;
  TEMP13 : INT ;
  TEMP14 : INT ;
  TEMP15 : INT ;
  TEMP16 : INT ;
  TEMP17 : INT ;
  TEMP18 : INT ;
END_VAR
BEGIN
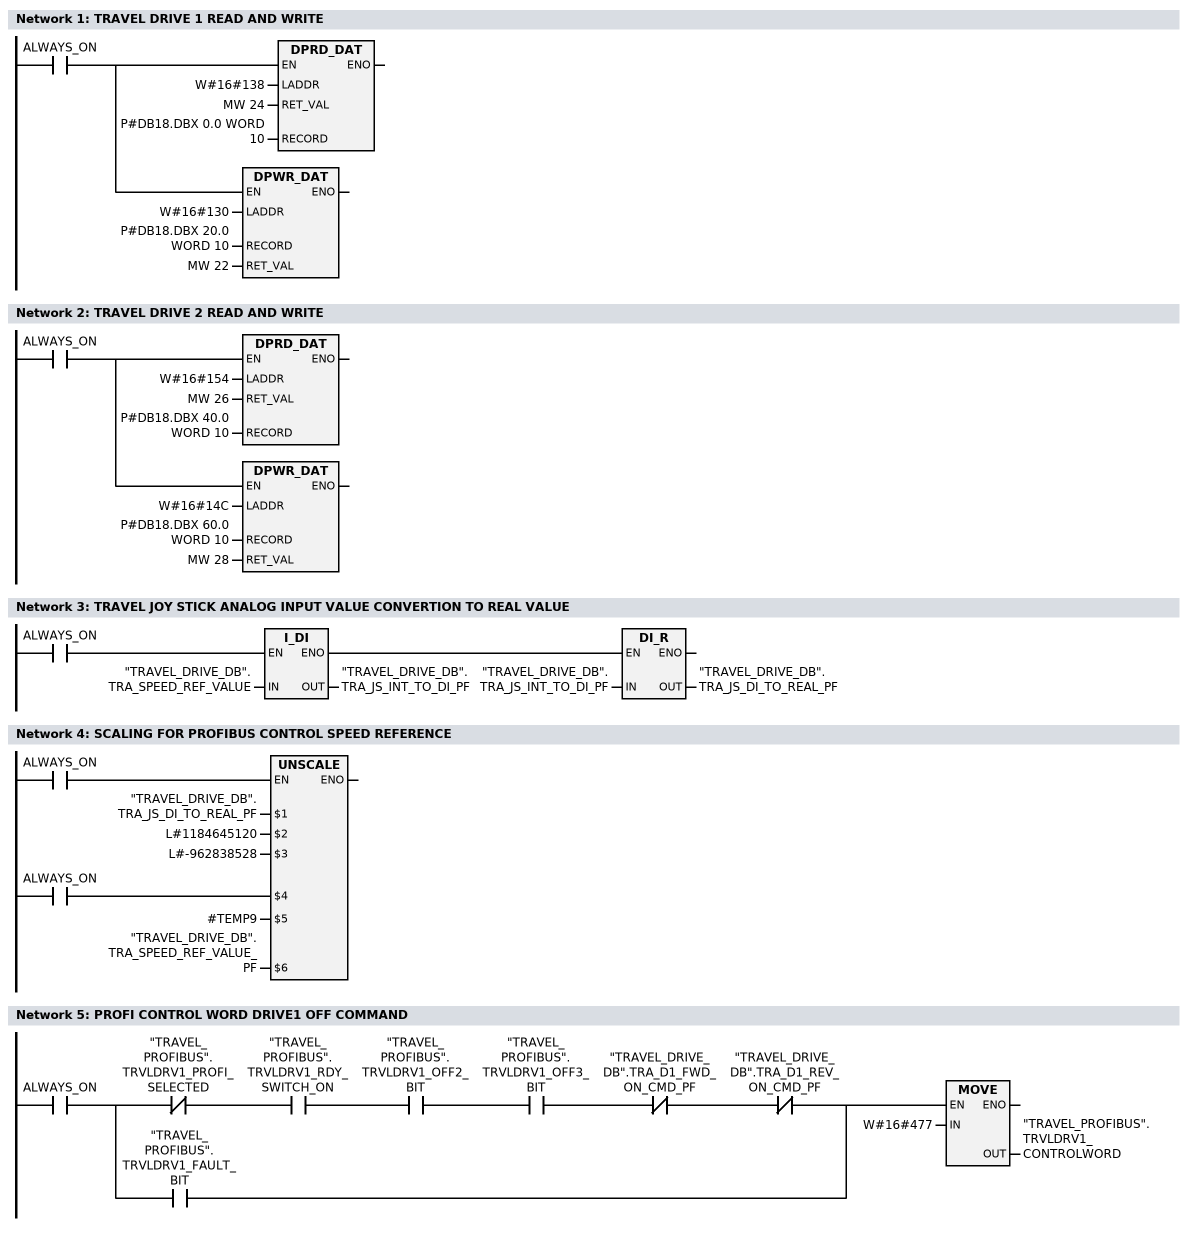
NETWORK
TITLE = TRAVEL DRIVE 1 READ AND WRITE 
      A     "ALWAYS_ON";
      =     L 36.0;
      A     L 36.0;
      JNB   _001;
      CALL  "DPRD_DAT" (
           LADDR                    := W#16#138,
           RET_VAL                  := MW 24,
           RECORD                   := P#DB18.DBX 0.0 WORD 10);
_001: NOP   0;
      A     L 36.0;
      JNB   _002;
      CALL  "DPWR_DAT" (
           LADDR                    := W#16#130,
           RECORD                   := P#DB18.DBX 20.0 WORD 10,
           RET_VAL                  := MW 22);
_002: NOP   0;
NETWORK
TITLE = TRAVEL DRIVE 2 READ AND WRITE 
      A     "ALWAYS_ON";
      =     L 36.0;
      A     L 36.0;
      JNB   _003;
      CALL  "DPRD_DAT" (
           LADDR                    := W#16#154,
           RET_VAL                  := MW 26,
           RECORD                   := P#DB18.DBX 40.0 WORD 10);
_003: NOP   0;
      A     L 36.0;
      JNB   _004;
      CALL  "DPWR_DAT" (
           LADDR                    := W#16#14C,
           RECORD                   := P#DB18.DBX 60.0 WORD 10,
           RET_VAL                  := MW 28);
_004: NOP   0;
NETWORK
TITLE = TRAVEL JOY STICK ANALOG INPUT VALUE CONVERTION TO REAL VALUE
//TRAVEL DRIVE JOY STICK ANALOG INPUT VALUE CONVERTION TO REAL VALUE
      A(;
      A     "ALWAYS_ON";
      JNB   _005;
      L     "TRAVEL_DRIVE_DB".TRA_SPEED_REF_VALUE;
      ITD;
      T     "TRAVEL_DRIVE_DB".TRA_JS_INT_TO_DI_PF;
      SET;
      SAVE;
      CLR;
_005: A     BR;
      );
      JNB   _006;
      L     "TRAVEL_DRIVE_DB".TRA_JS_INT_TO_DI_PF;
      DTR;
      T     "TRAVEL_DRIVE_DB".TRA_JS_DI_TO_REAL_PF;
_006: NOP   0;
NETWORK
TITLE = SCALING FOR PROFIBUS CONTROL SPEED REFERENCE
      A     "ALWAYS_ON";
      =     L 36.0;
      BLD   103;
      A     "ALWAYS_ON";
      JNB   _007;
      CALL  "UNSCALE" (
           $1                       := "TRAVEL_DRIVE_DB".TRA_JS_DI_TO_REAL_PF,
           $2                       := L#1184645120,
           $3                       := L#-962838528,
           $4                       := L 36.0,
           $5                       := #TEMP9,
           $6                       := "TRAVEL_DRIVE_DB".TRA_SPEED_REF_VALUE_PF);
_007: NOP   0;
NETWORK
TITLE = PROFI CONTROL WORD DRIVE1 OFF COMMAND
      A     "ALWAYS_ON";
      A(;
      AN    "TRAVEL_PROFIBUS".TRVLDRV1_PROFI_SELECTED;
      A     "TRAVEL_PROFIBUS".TRVLDRV1_RDY_SWITCH_ON;
      A     "TRAVEL_PROFIBUS".TRVLDRV1_OFF2_BIT;
      A     "TRAVEL_PROFIBUS".TRVLDRV1_OFF3_BIT;
      AN    "TRAVEL_DRIVE_DB".TRA_D1_FWD_ON_CMD_PF;
      AN    "TRAVEL_DRIVE_DB".TRA_D1_REV_ON_CMD_PF;
      O     "TRAVEL_PROFIBUS".TRVLDRV1_FAULT_BIT;
      );
      JNB   _008;
      L     W#16#477;
      T     "TRAVEL_PROFIBUS".TRVLDRV1_CONTROLWORD;
_008: NOP   0;
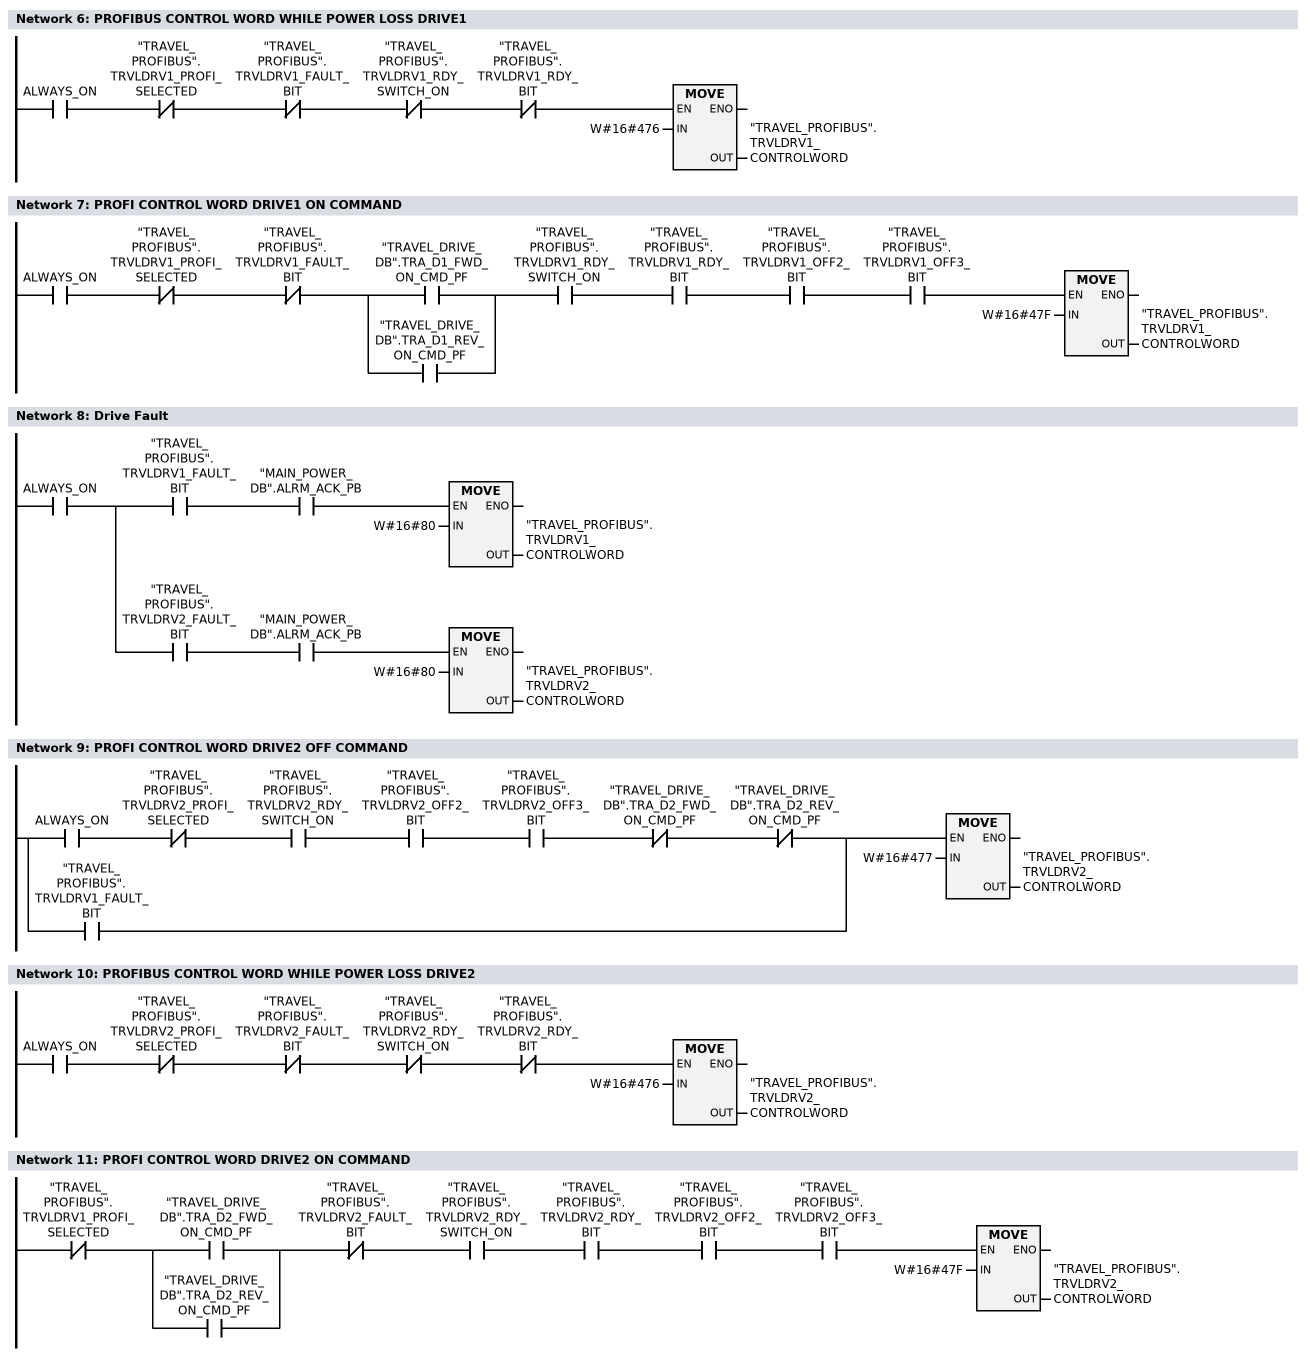
NETWORK
TITLE = PROFIBUS CONTROL WORD WHILE POWER LOSS DRIVE1
      A     "ALWAYS_ON";
      AN    "TRAVEL_PROFIBUS".TRVLDRV1_PROFI_SELECTED;
      AN    "TRAVEL_PROFIBUS".TRVLDRV1_FAULT_BIT;
      AN    "TRAVEL_PROFIBUS".TRVLDRV1_RDY_SWITCH_ON;
      AN    "TRAVEL_PROFIBUS".TRVLDRV1_RDY_BIT;
      JNB   _009;
      L     W#16#476;
      T     "TRAVEL_PROFIBUS".TRVLDRV1_CONTROLWORD;
_009: NOP   0;
NETWORK
TITLE = PROFI CONTROL WORD DRIVE1 ON COMMAND
      A     "ALWAYS_ON";
      AN    "TRAVEL_PROFIBUS".TRVLDRV1_PROFI_SELECTED;
      AN    "TRAVEL_PROFIBUS".TRVLDRV1_FAULT_BIT;
      A(;
      O     "TRAVEL_DRIVE_DB".TRA_D1_FWD_ON_CMD_PF;
      O     "TRAVEL_DRIVE_DB".TRA_D1_REV_ON_CMD_PF;
      );
      A     "TRAVEL_PROFIBUS".TRVLDRV1_RDY_SWITCH_ON;
      A     "TRAVEL_PROFIBUS".TRVLDRV1_RDY_BIT;
      A     "TRAVEL_PROFIBUS".TRVLDRV1_OFF2_BIT;
      A     "TRAVEL_PROFIBUS".TRVLDRV1_OFF3_BIT;
      JNB   _00a;
      L     W#16#47F;
      T     "TRAVEL_PROFIBUS".TRVLDRV1_CONTROLWORD;
_00a: NOP   0;
NETWORK
TITLE = Drive Fault
      A     "ALWAYS_ON";
      =     L 36.0;
      A     L 36.0;
      A     "TRAVEL_PROFIBUS".TRVLDRV1_FAULT_BIT;
      A     "MAIN_POWER_DB".ALRM_ACK_PB;
      JNB   _00b;
      L     W#16#80;
      T     "TRAVEL_PROFIBUS".TRVLDRV1_CONTROLWORD;
_00b: NOP   0;
      A     L 36.0;
      A     "TRAVEL_PROFIBUS".TRVLDRV2_FAULT_BIT;
      A     "MAIN_POWER_DB".ALRM_ACK_PB;
      JNB   _00c;
      L     W#16#80;
      T     "TRAVEL_PROFIBUS".TRVLDRV2_CONTROLWORD;
_00c: NOP   0;
NETWORK
TITLE = PROFI CONTROL WORD DRIVE2 OFF COMMAND
      A(;
      A     "ALWAYS_ON";
      AN    "TRAVEL_PROFIBUS".TRVLDRV2_PROFI_SELECTED;
      A     "TRAVEL_PROFIBUS".TRVLDRV2_RDY_SWITCH_ON;
      A     "TRAVEL_PROFIBUS".TRVLDRV2_OFF2_BIT;
      A     "TRAVEL_PROFIBUS".TRVLDRV2_OFF3_BIT;
      AN    "TRAVEL_DRIVE_DB".TRA_D2_FWD_ON_CMD_PF;
      AN    "TRAVEL_DRIVE_DB".TRA_D2_REV_ON_CMD_PF;
      O     "TRAVEL_PROFIBUS".TRVLDRV1_FAULT_BIT;
      );
      JNB   _00d;
      L     W#16#477;
      T     "TRAVEL_PROFIBUS".TRVLDRV2_CONTROLWORD;
_00d: NOP   0;
NETWORK
TITLE = PROFIBUS CONTROL WORD WHILE POWER LOSS DRIVE2
      A     "ALWAYS_ON";
      AN    "TRAVEL_PROFIBUS".TRVLDRV2_PROFI_SELECTED;
      AN    "TRAVEL_PROFIBUS".TRVLDRV2_FAULT_BIT;
      AN    "TRAVEL_PROFIBUS".TRVLDRV2_RDY_SWITCH_ON;
      AN    "TRAVEL_PROFIBUS".TRVLDRV2_RDY_BIT;
      JNB   _00e;
      L     W#16#476;
      T     "TRAVEL_PROFIBUS".TRVLDRV2_CONTROLWORD;
_00e: NOP   0;
NETWORK
TITLE = PROFI CONTROL WORD DRIVE2 ON COMMAND
      AN    "TRAVEL_PROFIBUS".TRVLDRV1_PROFI_SELECTED;
      A(;
      O     "TRAVEL_DRIVE_DB".TRA_D2_FWD_ON_CMD_PF;
      O     "TRAVEL_DRIVE_DB".TRA_D2_REV_ON_CMD_PF;
      );
      AN    "TRAVEL_PROFIBUS".TRVLDRV2_FAULT_BIT;
      A     "TRAVEL_PROFIBUS".TRVLDRV2_RDY_SWITCH_ON;
      A     "TRAVEL_PROFIBUS".TRVLDRV2_RDY_BIT;
      A     "TRAVEL_PROFIBUS".TRVLDRV2_OFF2_BIT;
      A     "TRAVEL_PROFIBUS".TRVLDRV2_OFF3_BIT;
      JNB   _00f;
      L     W#16#47F;
      T     "TRAVEL_PROFIBUS".TRVLDRV2_CONTROLWORD;
_00f: NOP   0;
